# B&R Automation Studio project Palletizer
Automation Studio 4.9

## Logical view

Binary libraries used (declarations not repeated): operator, runtime, astime, AsIecCon, standard, AsArLog, AsBrStr, AsTCP, MTBasics, brsystem, MTTypes, sys_lib, Acp10man, Acp10par, NcGlobal

### Global.var - Global variables
```iecst
(*Feeder*)
(*Inputs*)
VAR
	ResetButton : BOOL;
	laser_sensor_IR : BOOL;
	laser_sensor_2_IR : BOOL;
	carriage_2_AXIS : REAL;
	carriage_2_RCHD : BOOL;
	turnpusher_LBK : BOOL;
	turnpusher_LFR : BOOL;
	pusher_LBK : BOOL;
	pusher_LFR : BOOL;
END_VAR
(*Outputs*)
VAR
	pusher_FW : BOOL;
	conveyor_if_FWD : BOOL;
	conveyor_turn1_FWD : BOOL;
	conveyor_end_FWD : BOOL;
	carrige_2_TGT_POS : REAL;
	turnpusher_FWD : BOOL;
	turnpusher_BWD : BOOL;
END_VAR
(*GenericDevice Feeder requests*)
VAR
	conveyor_if_enable_request : BOOL;
	conveyor_if_disable_request : BOOL;
	conveyor_turn1_enable_request : BOOL;
	conveyor_turn1_disable_request : BOOL;
	conveyor_end_enable_request : BOOL;
	conveyor_end_disable_request : BOOL;
	pusher_enable_request : BOOL;
	pusher_disable_request : BOOL;
	turnpusher_enable_request : BOOL;
	turnpusher_disable_request : BOOL;
	OperationType : INT := 0;
END_VAR
(*Feeder-Main communication variable*)
VAR
	StartMachine : BOOL;
	FeederInitDone : BOOL;
	FeederStart : BOOL;
	FeederHomed : BOOL;
	FeederReady : BOOL;
	FeederEnable : BOOL;
	FeederIsReady : BOOL;
	CraneEnable : BOOL;
	CraneIsReady : BOOL;
	CraneStart : BOOL;
	FeederStop : BOOL;
	vacuum_box_crane_VACUUM : BOOL;
	box_crane_AXIS : REAL;
	gantry_crane_AXIS : REAL;
	gantry_crane_TGT_POS : REAL;
	box_crane_TGT_POS : REAL;
	cardboard_TRIG : BOOL;
	vaccum_box_crane_GRIP : BOOL;
	slide_rail_right_EN : BOOL;
	pusher_z_EN : BOOL;
	pusher_x_EN : BOOL;
END_VAR
(*Crane-Main communication variable*)
VAR
	CraneStop : BOOL;
	CraneHomed : BOOL;
	FeederHoming : BOOL;
	Trigger : BOOL;
	autoreset : BOOL;
	EmergencyStop : BOOL;
	vacuum_box_crane_GRIP : BOOL;
	MainEnable : BOOL;
	MainStart : BOOL;
	PalletHandlerEnable : BOOL;
	pallet_conveyor_2_ACT_VEL : REAL;
	PalletHandlerStart : BOOL;
	pallet_light_barrier_2_IR : BOOL;
	pallet_light_barrier_1_IR : BOOL;
	pallet_conveyor_1_FWD : BOOL;
	pallet_fork_left_EN : BOOL;
	pallet_fork_left_FB : BOOL;
	pallet_lifter_AXIS : REAL;
	pallet_lifter_TGT_POS : REAL;
	PalletHandlerIsReady : BOOL;
	cartboard_TRIG : BOOL;
	PusherXActuatorFaultE : BOOL;
	PusherXDisableSensorFaultE : BOOL;
	PusherXEnableSensorFaultE : BOOL;
	PusherZActuatorFaultE : BOOL;
	PusherZDisableSensorFaultE : BOOL;
	PusherZEnableSensorFaultE : BOOL;
	SlideRailRightActuatorFaultE : BOOL;
	SlideRailRightDisableFaultE : BOOL;
	SlideRailRightEnableFaultE : BOOL;
	VacuumBoxCraneActuatorFaultE : BOOL;
	VacuumBoxCraneDisableFaultE : BOOL;
	VacuumBoxCraneEnableFaultE : BOOL;
	CardboardActuatorFaultE : BOOL;
	CardboardDisableFaultE : BOOL;
	BoxCraneFaultSignalE : BOOL;
	GantryCraneFaultSignalE : BOOL;
	CardboardEnableFaultE : BOOL;
	TurnpusherActuatorFaultE : BOOL;
	TurnpusherDisableSensorFaultE : BOOL;
	TurnpusherEnableSensorFaultE : BOOL;
	PusherActuatorFaultE : BOOL;
	PusherDisableSensorFaultE : BOOL;
	PusherEnableSensorFaultE : BOOL;
	ConveyorIfActuatorFaultE : BOOL;
	ConveyorIfDisableSensorFaultE : BOOL;
	ConveyorIfEnableSensorFaultE : BOOL;
	ConveyorTurn1ActuatorFaultE : BOOL;
	ConveyorTurn1DisableSensorFaultE : BOOL;
	ConveyorTurn1EnableSensorFaultE : BOOL;
	ConveyorEndActuatorFaultE : BOOL;
	ConveyorEndDisableSensorFaultE : BOOL;
	ConveyorEndEnableSensorFaultE : BOOL;
	CarriagePositionFaultSignalE : BOOL;
	PalletForkActuatorFaultE : BOOL;
	PalletForkDisableSensorFaultE : BOOL;
	PalletForkEnableSensorFaultE : BOOL;
	PalletLifterFaultSignalE : BOOL;
	PalletConv1ActuatorFaultE : BOOL;
	PalletConv1DisableSensorFaultE : BOOL;
	PalletConv1SensorFaultE : BOOL;
	PalletConv2FaultSignalE : BOOL;
	LaserSensor2IRFault : BOOL;
	Var2 : BOOL;
	Var1 : BOOL;
	LogFile : STRING[3000];
	MainMessage : STRING[30];
	OnPhaseStop : BOOL;
	ImmediateStop : BOOL;
	ImmediateStopButton : BOOL;
	EmergencyStopButton : BOOL;
	OnPhaseStopPerforming : BOOL;
	OnPhaseStopButton : BOOL;
	laser_sensor_IR_enabled : BOOL;
	pallet_light_barrier_enabled : BOOL;
	laser_sensor_2_IR_enabled : BOOL;
	pallet_light_barrier2_enabled : BOOL;
	InfoCarousel : STRING[20];
	HomeButton : BOOL;
	ErrorButton : BOOL;
	OrangeLight : BOOL;
	YellowLight : BOOL;
	ResetEnable : BOOL;
	WhiteLight : BOOL;
	BlueLight : BOOL;
	GreenLight : BOOL;
	RedLight : BOOL;
	SimPusherActuatorFaultE : BOOL;
	SimPusherDisableSensorFaultE : BOOL;
	SimBoxCraneFaultSignalE : BOOL;
	SimVacuumBoxCraneActuatorFaultE : BOOL;
	SimPalletForkActuatorFaultE : BOOL;
	SimPalletForkEnableSensorFaultE : BOOL;
	OperationTypeString : STRING[20];
	CounterPallet : INT;
END_VAR
```

### Package Logical/Libraries - Global libraries

### Library Logical/Libraries/GenericDev (IEC)

#### Types.typ - Exported data types
```iecst
TYPE
	GenericDeviceStateType :
		(
		DeviceDisabledState,
		DeviceEnablePhaseState,
		DeviceEnabledState,
		DeviceDisablePhaseState
		);
END_TYPE
```

#### Constants.var - Exported constants
```iecst
VAR CONSTANT
	INIT : INT := 0;
	RUN : INT := 1;
	ENABLED : INT := 2;
	STOP : INT := 3;
	DEVICE_WITHOUT_FEEDBACK : INT := 2#01000000;
	DEVICE_WITH_ENABLE_FEEDBACK : INT := 2#00010000;
	DEVICE_WITH_DISABLE_FEEDBACK : INT := 2#00100000;
	DEVICE_WITH_DOUBLE_FEEDBACK : INT := 2#00110000;
	DEVICE_WITH_SINGLE_ACTUATION : INT := 2#00000001;
	DEVICE_WITH_DOUBLE_ACTUATION : INT := 2#00000011;
	DEVICE_IMMEDIATE_STOP_AUTOMATIC : INT := 2#10000000;
	DEVICE_WITH_DA_NO_RETAIN : INT := 2#00000010;
	DEVICE_FEEDBACK_MASK : INT := 2#01110000;
	DEVICE_STOP_MASK : INT := 2#10000000;
	DEVICE_ACTUATION_MASK : INT := 2#00001111;
END_VAR
```

#### GenericDev.fun - Exported functions and function blocks
```iecst
FUNCTION_BLOCK GenericDevice_FB
	VAR_INPUT
		DeviceOperation : INT;
		DeviceType : INT;
		DeviceEnabledSensor : BOOL;
		DeviceDisabledSensor : BOOL;
		DeviceClock : BOOL;
		DeviceEnableTime : INT;
		DeviceDisableTime : INT;
		DeviceDiagnosticsEnabled : BOOL;
		DeviceEnablePreset : BOOL;
		ImmediateStop : BOOL;
	END_VAR
	VAR_OUTPUT
		EnableDevice : BOOL;
		DisableDevice : BOOL;
		DeviceEnabledSensorFault : BOOL;
		DeviceDisabledSensorFault : BOOL;
		DeviceActuatorFault : BOOL;
		DeviceFault : BOOL;
		DeviceNotInitialized : BOOL;
	END_VAR
	VAR_IN_OUT
		DeviceEnableRequest : BOOL;
		DeviceDisableRequest : BOOL;
	END_VAR
	VAR
		DeviceState : GenericDeviceStateType;
		DeviceTimer : INT;
		DeviceTimeout : BOOL;
		DeviceEnabled : BOOL;
		DeviceDisabled : BOOL;
		OldEnableDevice : BOOL;
		Condition : BOOL;
	END_VAR
END_FUNCTION_BLOCK
```

#### GenericDevice_FB.st
```iecst
(*Generic Device function block implementation (See Slide Generic Device)*)
FUNCTION_BLOCK GenericDevice_FB

    // Device clock handler
	IF (DeviceClock AND (DeviceTimer > 0)) THEN
		DeviceTimer := DeviceTimer - 1;
	END_IF;

	// Device sensors handler
	CASE (DeviceType AND DEVICE_FEEDBACK_MASK) OF
		DEVICE_WITH_DISABLE_FEEDBACK:

			DeviceDisabled := DeviceDisabledSensor;

			DeviceEnabled := NOT DeviceDisabled AND
				((DeviceState = DeviceEnabledState) OR
				((DeviceState = DeviceEnablePhaseState) AND DeviceTimeout));

		DEVICE_WITH_ENABLE_FEEDBACK:

			DeviceEnabled := DeviceEnabledSensor;

			DeviceDisabled := NOT DeviceEnabled AND
				((DeviceState = DeviceDisabledState) OR
				((DeviceState = DeviceDisablePhaseState) AND DeviceTimeout));

		DEVICE_WITH_DOUBLE_FEEDBACK:

			DeviceEnabled := DeviceEnabledSensor;

			DeviceDisabled := DeviceDisabledSensor;

		DEVICE_WITHOUT_FEEDBACK:

			DeviceEnabled := (DeviceState = DeviceEnabledState) OR ((DeviceState = DeviceEnablePhaseState) AND DeviceTimeout);

			DeviceDisabled := (DeviceState = DeviceDisabledState) OR ((DeviceState = DeviceDisablePhaseState) AND DeviceTimeout);

	END_CASE;

	// Initialization handler
	IF DeviceOperation = INIT THEN
		CASE (DeviceType AND DEVICE_FEEDBACK_MASK) OF
			DEVICE_WITH_ENABLE_FEEDBACK:
				DeviceDisabled := NOT DeviceEnabled;

			DEVICE_WITH_DISABLE_FEEDBACK:
				DeviceEnabled := NOT DeviceDisabled;

			DEVICE_WITHOUT_FEEDBACK:
				DeviceEnabled := DeviceEnablePreset;
				DeviceDisabled := NOT DeviceEnabled;
		END_CASE;

		DeviceEnableRequest := FALSE;
		DeviceDisableRequest := FALSE;

		IF DeviceEnablePreset THEN
			EnableDevice := TRUE;
			DeviceTimer := DeviceEnableTime;
			IF NOT (DeviceDisabled AND DeviceEnabled) THEN
				DeviceState := DeviceEnablePhaseState;
			ELSE
				DeviceState := DeviceEnabledState;
			END_IF;
			DeviceNotInitialized := NOT DeviceEnabled OR DeviceDisabled;
		ELSE
			EnableDevice := FALSE;
			DeviceTimer := DeviceDisableTime;
			IF NOT (DeviceDisabled AND DeviceEnabled) THEN
				DeviceState := DeviceDisablePhaseState;
			ELSE
				DeviceState := DeviceDisabledState;
			END_IF;
			DeviceNotInitialized := DeviceEnabled OR NOT DeviceDisabled;
		END_IF;
	END_IF;

	// Device control handler (slide 8-9)
	CASE DeviceState OF
		DeviceDisabledState:
			DeviceDisableRequest := FALSE;
			IF (DeviceEnableRequest) THEN
				EnableDevice := TRUE;
				DeviceTimer := DeviceEnableTime;
				DeviceState := DeviceEnablePhaseState;
			END_IF;

		DeviceEnablePhaseState:
			IF (DeviceDisableRequest) THEN
				DeviceEnableRequest := FALSE;
				EnableDevice := FALSE;
				DeviceTimer := DeviceDisableTime;
				DeviceState := DeviceDisablePhaseState;
			END_IF;
			IF (DeviceEnabled) THEN
				DeviceEnableRequest := FALSE;
				//DeviceTimer := 0;
				DeviceState := DeviceEnabledState;
			END_IF;

		DeviceEnabledState:
			DeviceEnableRequest := FALSE;
			IF (DeviceDisableRequest) THEN
				EnableDevice := FALSE;
				DeviceTimer := DeviceDisableTime;
				DeviceState := DeviceDisablePhaseState;
			END_IF;

		DeviceDisablePhaseState:
			IF (DeviceEnableRequest) THEN
				DeviceDisableRequest := FALSE;
				EnableDevice := TRUE;
				DeviceTimer := DeviceEnableTime;
				DeviceState := DeviceEnablePhaseState;
			END_IF;
			IF (DeviceDisabled) THEN
				DeviceDisableRequest := FALSE;
				//DeviceTimer := 0;
				DeviceState := DeviceDisabledState;
			END_IF;
	END_CASE;

	// Device diagnostics handler (slide 26)
	DeviceTimeout := (DeviceTimer = 0);
	IF DeviceDiagnosticsEnabled AND NOT ImmediateStop AND (DeviceType AND DEVICE_FEEDBACK_MASK) <> DEVICE_WITHOUT_FEEDBACK THEN
		CASE (DeviceType AND DEVICE_FEEDBACK_MASK) OF
			DEVICE_WITH_DISABLE_FEEDBACK:

				DeviceDisabledSensorFault :=
				(NOT EnableDevice AND NOT DeviceDisabled AND NOT DeviceEnabled) AND DeviceTimeout;

				DeviceActuatorFault :=
				(EnableDevice AND DeviceDisabled AND NOT DeviceEnabled) AND DeviceTimeout;

			DEVICE_WITH_ENABLE_FEEDBACK:

				DeviceEnabledSensorFault :=
				(EnableDevice AND NOT DeviceDisabled AND NOT DeviceEnabled) AND DeviceTimeout;

				DeviceActuatorFault :=
				(NOT EnableDevice AND NOT DeviceDisabled AND DeviceEnabled) AND DeviceTimeout;

			DEVICE_WITH_DOUBLE_FEEDBACK:

				DeviceDisabledSensorFault :=
				((NOT EnableDevice AND NOT DeviceDisabled AND NOT DeviceEnabled) OR
				(EnableDevice AND DeviceDisabled AND DeviceEnabled)) AND DeviceTimeout;

				DeviceEnabledSensorFault :=
				((NOT EnableDevice AND DeviceDisabled AND DeviceEnabled) OR
				(EnableDevice AND NOT DeviceDisabled AND NOT DeviceEnabled)) AND DeviceTimeout;

				DeviceActuatorFault :=
				((NOT EnableDevice AND NOT DeviceDisabled AND DeviceEnabled) OR
				(EnableDevice AND DeviceDisabled AND NOT DeviceEnabled)) AND DeviceTimeout;

		END_CASE;

		DeviceFault := DeviceDisabledSensorFault OR DeviceEnabledSensorFault OR DeviceActuatorFault;
	END_IF

	IF (DeviceType AND DEVICE_STOP_MASK) = DEVICE_IMMEDIATE_STOP_AUTOMATIC AND ImmediateStop AND NOT Condition THEN
		OldEnableDevice := EnableDevice;
		EnableDevice := FALSE;
		Condition := TRUE;
	ELSIF Condition AND NOT ImmediateStop THEN
		EnableDevice := OldEnableDevice;
		Condition := FALSE;
	END_IF

	// Device actuators handler (correct from slides)
	CASE (DeviceType AND DEVICE_ACTUATION_MASK) OF
		DEVICE_WITH_DOUBLE_ACTUATION:
			DisableDevice := NOT EnableDevice;

		DEVICE_WITH_DA_NO_RETAIN:
			EnableDevice := EnableDevice AND (DeviceState = DeviceEnablePhaseState);
			DisableDevice := NOT EnableDevice AND(DeviceState = DeviceDisablePhaseState);
	END_CASE;

END_FUNCTION_BLOCK
```

### Library Logical/Libraries/GenericAx (IEC)

#### Types.typ - Exported data types
```iecst
TYPE
	GenericAxisStateType :
		(
		CheckCommand,
		WaitTargetPosition,
		WaitTargetVelocity,
		FaultState,
		StopEmergencyState,
		WaitForStop
		);
END_TYPE
```

#### Constants.var - Exported constants
```iecst
VAR CONSTANT
	IDLE : WORD := 0;
	CHANGE_VELOCITY : WORD := 1;
	CHANGE_POSITION : WORD := 2;
	EMERGENCY_STOP_REQUEST : WORD := 3;
	IMMEDIATE_STOP_REQUEST : WORD := 4;
END_VAR
```

#### GenericAx.fun - Exported functions and function blocks
```iecst
{REDUND_ERROR} FUNCTION_BLOCK GenericAxis (*TODO: Add your comment here*) (*$GROUP=User,$CAT=User,$GROUPICON=User.png,$CATICON=User.png*)
	VAR_INPUT
		Command : {REDUND_UNREPLICABLE} WORD := 6;
		ActualPosition : REAL;
		ActualVelocity : REAL;
		NewSetPoint : REAL;
		DeviceTimer : UDINT;
		TGT_SENSOR : BOOL;
		Reset : BOOL;
	END_VAR
	VAR_OUTPUT
		TargetVelocity : REAL;
		TargetPosition : REAL;
		InPosition : BOOL;
		InVelocity : BOOL;
		DeviceFault : BOOL;
	END_VAR
	VAR
		AxisState : GenericAxisStateType;
		Timer : UDINT;
	END_VAR
END_FUNCTION_BLOCK
```

#### GenericAxis.st
```iecst
(* GenericAxis function block *)
FUNCTION_BLOCK GenericAxis

	CASE AxisState OF

		CheckCommand:
			IF Command = CHANGE_POSITION THEN
				IF TargetPosition <> NewSetPoint THEN
					TargetPosition := NewSetPoint;
					InPosition := FALSE;
					Timer := DeviceTimer;
					AxisState := WaitTargetPosition;
				END_IF

			ELSIF Command = CHANGE_VELOCITY THEN
				IF TargetVelocity <> NewSetPoint THEN
					TargetVelocity := NewSetPoint;
					InVelocity := FALSE;
					Timer := DeviceTimer;
					AxisState := WaitTargetVelocity;
				END_IF

			ELSIF Command = IMMEDIATE_STOP_REQUEST OR Command = EMERGENCY_STOP_REQUEST THEN
				TargetPosition := ActualPosition;
				TargetVelocity := 0;
				AxisState := StopEmergencyState;

			ELSIF Command = IDLE THEN
				IF (ActualPosition = TargetPosition AND TGT_SENSOR) THEN
					InPosition := TRUE;
				ELSE
					InPosition := FALSE;
				END_IF
				IF (ActualVelocity = TargetVelocity) THEN
					InVelocity := TRUE;
				ELSE
					InVelocity := FALSE;
				END_IF
				Timer := DeviceTimer;
				DeviceFault := FALSE;
			END_IF

		WaitTargetPosition:
			IF  Command = IMMEDIATE_STOP_REQUEST OR Command = EMERGENCY_STOP_REQUEST THEN
				TargetPosition := ActualPosition;
				TargetVelocity := 0;
				AxisState := StopEmergencyState;
			ELSIF (ActualPosition = TargetPosition AND TGT_SENSOR) THEN
				InPosition := TRUE;
				AxisState := CheckCommand;
			END_IF

			Timer := Timer - 1;
			IF Timer = 0 THEN
				DeviceFault := TRUE;
				AxisState := FaultState;
			END_IF

		WaitTargetVelocity:
			IF  Command = IMMEDIATE_STOP_REQUEST OR Command = EMERGENCY_STOP_REQUEST THEN
				TargetVelocity := 0;
				AxisState := StopEmergencyState;

			ELSIF ActualVelocity = TargetVelocity THEN
				InVelocity := TRUE;
				AxisState := CheckCommand;
			END_IF

			Timer := Timer - 1;
			IF Timer = 0 THEN
				DeviceFault := TRUE;
				AxisState := FaultState;
			END_IF

		StopEmergencyState:
			IF Command <> IMMEDIATE_STOP_REQUEST AND Command <> EMERGENCY_STOP_REQUEST THEN
				InPosition := FALSE;
				InVelocity := FALSE;
				AxisState := CheckCommand;
			END_IF

		FaultState:
			IF Reset THEN
				DeviceFault := FALSE;
				AxisState := CheckCommand;
			END_IF

	END_CASE;

END_FUNCTION_BLOCK
```

### Library Logical/Libraries/Signal_lib (IEC)

#### Constants.var - Exported constants
```iecst
(*OUTPUTS*)
VAR CONSTANT
	NONE : DWORD := 16#0000;
	EMERGENCY_STOP : DWORD := 16#0001;
	ON_PHASE_STOP : DWORD := 16#0010;
	IMMEDIATE_STOP : DWORD := 16#0100; (*Operation types for the Signal Manager*)
	START_CONFIGURATION : USINT := 1;
	CONFIGURATION : USINT := 2;
	START_GENERATION : USINT := 3;
	MESSAGES_GENERATION : USINT := 5;
	GENERATION : USINT := 4; (*SignalCode bitmap*)
	INFORMATION : USINT := 1;
	ANOMALY : USINT := 2;
	WARNING : USINT := 3;
	ALARM : USINT := 4; (*masks for the SiglaCode*)
	DISPLAY_LOG : USINT := 8;
	SIGNAL_TYPE_MASK : USINT := 7;
	SIGNAL_LOG_MASK : USINT := 8;
END_VAR
```

#### Signal_lib.fun - Exported functions and function blocks
```iecst
{REDUND_ERROR} FUNCTION_BLOCK SignalManagement_FB (*TODO: Add your comment here*) (*$GROUP=User,$CAT=User,$GROUPICON=User.png,$CATICON=User.png*)
	VAR_INPUT
		OperationType : INT;
		SignalType : INT; (* bit configuration for the signal*)
		Reset : BOOL;
		KeyReset : BOOL;
		SignalOutput : DWORD; (* Output of the Signal if active*)
		ActivationSignal : {REDUND_UNREPLICABLE} BOOL;
		SignalCode : INT; (* Is the signal number in the priority list*)
		InputString : STRING[80];
	END_VAR
	VAR_OUTPUT
		MainMessage : STRING[30];
		LogFile : STRING[3000];
		SignalOutputs : DWORD; (*Output Signal codification*)
	END_VAR
	VAR
		LogBuffer : ARRAY[1..100] OF STRING[30];
		NumberOfAlarms : INT; (*Counters*)
		NumberOfAnomalies : INT;
		NumberOfWarnings : INT;
		NumberOfInformation : INT; (*Counters for Active Signals*)
		NumberOfActiveAlarms : INT;
		NumberOfActiveAnomalies : INT;
		NumberOfActiveWarning : INT;
		NumberOfActiveInformation : INT; (*Reset Management*)
	END_VAR
	VAR_OUTPUT
		ResetEnable : BOOL;
	END_VAR
	VAR
		ResetActivation : BOOL;
		AuxResetActivation : BOOL;
		Signals : ARRAY[1..100] OF BOOL; (*Signals management*)
		ActiveSignalCodes : ARRAY[1..100] OF INT;
		ResetOld : BOOL; (*Auxiliary variable*)
		KeyResetOld : BOOL;
		Index : INT;
		BaseIndex : INT;
		Condition : BOOL;
		i : INT;
	END_VAR
END_FUNCTION_BLOCK
```

#### SignalManagement_FB.st
```iecst
(* TODO: Add your comment here *)
FUNCTION_BLOCK SignalManagement_FB

	CASE OperationType OF
		START_CONFIGURATION:  (* Reset signals counts *)
			NumberOfAlarms := 0;
			NumberOfAnomalies := 0;
			NumberOfWarnings := 0;
			NumberOfInformation := 0;
			ResetEnable := FALSE;
		CONFIGURATION:
			(* counting signals *)
			CASE SignalType AND SIGNAL_TYPE_MASK OF
				ALARM:
					NumberOfAlarms := NumberOfAlarms + 1;
				ANOMALY:
					NumberOfAnomalies := NumberOfAnomalies + 1;
				WARNING:
					NumberOfWarnings := NumberOfWarnings + 1;
				INFORMATION:
					NumberOfInformation := NumberOfInformation + 1;
			END_CASE
		START_GENERATION:
			(* Prepare for generation *)
			ResetEnable := FALSE;
			SignalOutputs := NONE;
			ResetActivation := Reset AND NOT ResetOld;
			ResetOld := Reset;
			AuxResetActivation := KeyReset AND NOT KeyResetOld;
			KeyResetOld:= KeyReset;
			LogFile := '';
			MainMessage := '';

		GENERATION:
			CASE SignalType AND SIGNAL_TYPE_MASK OF
				ALARM:
					Index := NumberOfActiveAlarms;
					BaseIndex := 0;
					Condition := TRUE;
				ANOMALY:
					Index := NumberOfActiveAnomalies;
					BaseIndex := NumberOfAlarms;
					Condition := TRUE;
				WARNING:
					Index := NumberOfActiveWarning;
					BaseIndex := NumberOfAlarms + NumberOfAnomalies;
					Condition := FALSE;
				INFORMATION:
					Index := NumberOfActiveInformation;
					BaseIndex := NumberOfAlarms + NumberOfAnomalies + NumberOfWarnings;
					Condition := FALSE;
			END_CASE
			IF ActivationSignal AND NOT Signals[SignalCode] THEN
				Signals[SignalCode] := TRUE;
				Index := Index + 1;
				ActiveSignalCodes[BaseIndex + Index] := SignalCode;

				IF (SignalType AND SIGNAL_LOG_MASK) = DISPLAY_LOG THEN
					LogBuffer[SignalCode] := InputString;
				END_IF

			END_IF
			IF Condition AND Signals[SignalCode] AND NOT ActivationSignal AND (ActiveSignalCodes[BaseIndex + 1] = SignalCode) THEN
				ResetEnable := TRUE;
			END_IF

			IF (ResetActivation OR NOT Condition) AND Signals[SignalCode] AND NOT ActivationSignal AND (ActiveSignalCodes[BaseIndex + 1] = SignalCode) THEN
				Signals[SignalCode] := FALSE;
				FOR i := 2 TO Index DO
					ActiveSignalCodes[BaseIndex + i-1] := ActiveSignalCodes[BaseIndex + i];
				END_FOR;
				ActiveSignalCodes[BaseIndex + Index] := 0;
				Index :=  Index - 1;
				ResetActivation := FALSE; (* COMMENT THIS LINE TO GO BACK TO CUMULATIVE RESET *)

				IF (SignalType AND SIGNAL_LOG_MASK) = DISPLAY_LOG THEN
					LogBuffer[SignalCode] := ' ';
				END_IF

			END_IF
			CASE SignalType AND SIGNAL_TYPE_MASK OF
				ALARM:
					NumberOfActiveAlarms := Index;
				ANOMALY:
					NumberOfActiveAnomalies := Index;
				WARNING:
					NumberOfActiveWarning := Index;
				INFORMATION:
					NumberOfActiveInformation := Index;
			END_CASE
			IF Signals[SignalCode] THEN
				SignalOutputs := SignalOutputs OR SignalOutput;
			END_IF

		MESSAGES_GENERATION:

			LogFile := ' ';
			// ALARMS messages creation
			BaseIndex := 0;
			FOR i := 1 TO NumberOfActiveAlarms DO
				IF LogBuffer[ActiveSignalCodes[BaseIndex + i]] <> '' THEN
					LogFile := CONCAT(CONCAT(LogFile, CONCAT('ALARM : ',LogBuffer[ActiveSignalCodes[BaseIndex + i]])), ' \n ');
				END_IF
			END_FOR;

			// ANOMALIES messages creation
			BaseIndex := NumberOfAlarms;
			FOR i := 1 TO NumberOfActiveAnomalies DO
				IF LogBuffer[ActiveSignalCodes[BaseIndex + i]] <> '' THEN
					LogFile := CONCAT(CONCAT(LogFile,CONCAT('ANOMALY : ',LogBuffer[ActiveSignalCodes[BaseIndex + i]])), ' \n ');
				END_IF

			END_FOR;

			// WARNING messages creation
			BaseIndex := NumberOfAlarms + NumberOfAnomalies;
			FOR i := 1 TO NumberOfActiveWarning DO
				IF LogBuffer[ActiveSignalCodes[BaseIndex + i]] <> '' THEN
					LogFile := CONCAT(CONCAT(LogFile , CONCAT('WARNING : ',LogBuffer[ActiveSignalCodes[BaseIndex + i]])), ' \n ');
				END_IF
			END_FOR;

			// WARNING messages creation
			BaseIndex := NumberOfAlarms + NumberOfAnomalies + NumberOfWarnings;
			FOR i := 1 TO NumberOfActiveInformation DO
				IF LogBuffer[ActiveSignalCodes[BaseIndex + i]] <> '' THEN
					LogFile := CONCAT(CONCAT(LogFile , CONCAT('INFORMATION : ',LogBuffer[ActiveSignalCodes[BaseIndex + i]])), ' \n ');
				END_IF
			END_FOR;

			MainMessage := '';
			IF NumberOfActiveAlarms <> 0 THEN
				MainMessage := LogBuffer[ActiveSignalCodes[1]];
			ELSIF NumberOfActiveAnomalies <> 0 THEN
				MainMessage := LogBuffer[ActiveSignalCodes[NumberOfAlarms + 1]];
			ELSIF NumberOfActiveWarning <> 0 THEN
				MainMessage := LogBuffer[ActiveSignalCodes[NumberOfAlarms + NumberOfAnomalies + 1]];
			ELSIF NumberOfActiveInformation <> 0 THEN
				MainMessage := LogBuffer[ActiveSignalCodes[NumberOfAlarms + NumberOfAnomalies + NumberOfWarnings + 1]];
			END_IF

	END_CASE

END_FUNCTION_BLOCK
```

### Library Logical/Libraries/Filter (IEC)

#### Filter.fun - Exported functions and function blocks
```iecst
{REDUND_ERROR} {REDUND_UNREPLICABLE} FUNCTION_BLOCK filter_FB (*TODO: Add your comment here*) (*$GROUP=User,$CAT=User,$GROUPICON=User.png,$CATICON=User.png*)
	VAR_INPUT
		OperationType : {REDUND_UNREPLICABLE} INT;
		Clock : {REDUND_UNREPLICABLE} BOOL;
		Signal : {REDUND_UNREPLICABLE} BOOL;
		DeactivationDelay : {REDUND_UNREPLICABLE} INT;
		ActivationDelay : {REDUND_UNREPLICABLE} INT;
	END_VAR
	VAR_OUTPUT
		DelayedSignal : {REDUND_UNREPLICABLE} BOOL;
	END_VAR
	VAR
		Delay : {REDUND_UNREPLICABLE} INT;
	END_VAR
END_FUNCTION_BLOCK
```

#### filter_FB.st
```iecst
(* TODO: Add your comment here *)
FUNCTION_BLOCK filter_FB

	IF (OperationType = INIT) THEN
		Delay := 0;
	END_IF;

	IF (Clock AND (Delay > 0)) THEN
		Delay := Delay - 1;
	END_IF;

	IF  (Delay = 0) THEN
		DelayedSignal := Signal;
	END_IF;

	IF  (Signal = DelayedSignal) THEN
		IF  (Signal) THEN
			Delay := DeactivationDelay;
		ELSE
			Delay := ActivationDelay;
		END_IF;
	END_IF

END_FUNCTION_BLOCK
```

### Program Logical/MainCtrl (IEC)

#### Types.typ
```iecst
TYPE
	MainStateType :
		(
		Idle,
		Ready,
		Run,
		Init
		);
END_TYPE
```

#### Variables.var
```iecst
VAR
	MachineState : MainStateType;
END_VAR
```

#### Main.st
```iecst
PROGRAM _INIT

		MachineState := Idle;
END_PROGRAM

PROGRAM _CYCLIC

	CASE MachineState OF

		Idle:
			FeederEnable := FALSE;
			FeederHomed := FALSE;
			FeederStart := FALSE;

			IF StartMachine THEN
				FeederEnable := TRUE; (* sblocca alimentazione feeder *)
				MachineState := Init;
			END_IF

		Init:
			OperationType := INIT;
			StartMachine := FALSE;
			//FeederHomed := TRUE; (* manda homing feeder *)
			IF FeederHomed THEN // Need to add also the carriage
				FeederInitDone := TRUE;
			END_IF

			// Perform the same procedure for all the other 3 machines
			IF FeederInitDone THEN
				FeederReady := TRUE;  // States that all 3 machines are ready (now we consider only the feeder)
			END_IF

			IF FeederReady THEN
				MachineState := Ready;
			END_IF
		Ready:
			(* Attesa che anche crane e pallet handler siano ready, ora non li abbiamo *)
			OperationType := READY;
			IF StartMachine THEN
				FeederStart := TRUE;
				MachineState := Run;
			END_IF
		Run:
			OperationType := RUN;
			FeederHomed := FALSE;
			FeederEnable := TRUE;
			FeederStart := TRUE;

	END_CASE

END_PROGRAM

PROGRAM _EXIT
	(* Insert code here *)

END_PROGRAM
```

### MNG_Global.typ - Global data types
```iecst
(* 3d position *)

TYPE
	VEC3 : 	STRUCT
		x : REAL;
		y : REAL;
		z : REAL;
	END_STRUCT;
END_TYPE

(* position and orientation as an euler based pose *)

TYPE
	POSE6 : 	STRUCT
		x : REAL;
		y : REAL;
		z : REAL;
		a : REAL;
		b : REAL;
		c : REAL;
	END_STRUCT;
END_TYPE

(* position and orientation as a 4x4 matrix *)

TYPE
	TRAFO : 	STRUCT
		baseX : VEC3;
		fill0 : REAL;
		baseY : VEC3;
		fill1 : REAL;
		baseZ : VEC3;
		fill2 : REAL;
		origin : VEC3;
		fill3 : REAL;
	END_STRUCT;
END_TYPE
```

### Program Logical/FeederMachine (IEC)

#### Types.typ
```iecst
TYPE
	StateType :
		(
		Idle,
		EnableDone,
		Homing,
		HomingDone,
		WaitForStart,
		WaitForBoxes,
		PushBox,
		CheckSecondLaser,
		CheckPusherBackwardPosition,
		WaitBeforeCarriage,
		CarriageMidPush,
		CarriageTotalPush,
		CarriagePushBack,
		CarriageWaitForStart,
		EmergencyState,
		StopState,
		ImmediateStopState,
		CarriageMidPushDone,
		CarriageTotalPushDone
		);
END_TYPE
```

#### Variables.var
```iecst
VAR
	State : StateType;
END_VAR
(*Generic device variable interface for on/off actuations*)
(*conveyor_if*)
VAR
	conveyor_if : GenericDevice_FB;
END_VAR
VAR CONSTANT
	conveyor_if_enable_time : INT := 5;
	conveyor_if_disable_time : INT := 5;
END_VAR
VAR
	conveyor_if_enable_request : BOOL;
	conveyor_if_disable_request : BOOL;
END_VAR
(*conveyot_turn1*)
VAR
	conveyor_turn1 : GenericDevice_FB;
END_VAR
VAR CONSTANT
	conveyor_turn1_enable_time : INT := 5;
	conveyor_turn1_disable_time : INT := 5;
END_VAR
VAR
	conveyor_turn1_enable_request : BOOL;
	conveyor_turn1_disable_request : BOOL;
END_VAR
(*conveyor_end*)
VAR
	conveyor_end : GenericDevice_FB;
END_VAR
VAR CONSTANT
	conveyor_end_enable_time : INT := 5;
	conveyor_end_disable_time : INT := 5;
END_VAR
VAR
	conveyor_end_enable_request : BOOL;
	conveyor_end_disable_request : BOOL;
END_VAR
(*pusher*)
VAR
	pusher : GenericDevice_FB;
END_VAR
VAR CONSTANT
	pusher_enable_time : INT := 200;
	pusher_disable_time : INT := 200;
END_VAR
VAR
	pusher_enable_request : BOOL;
	pusher_disable_request : BOOL;
END_VAR
(*turnpusher*)
VAR
	turnpusher : GenericDevice_FB;
END_VAR
VAR CONSTANT
	turnpusher_enable_time : INT := 200;
	turnpusher_disable_time : INT := 200;
END_VAR
VAR
	turnpusher_enable_request : BOOL;
	turnpusher_disable_request : BOOL;
END_VAR
(*carriage*)
VAR
	carriage : GenericAxis;
	carriage_goal : REAL;
END_VAR
VAR CONSTANT
	carriage_timer : INT := 100;
END_VAR
VAR
	carriagePositionReached : BOOL;
	carriageSetPoint : USINT;
	carriage_homed : BOOL;
END_VAR
VAR CONSTANT
	HOME_POSITION : REAL := 0.0;
	CARRIAGE_MID_PUSH : REAL := 0.44;
	CARRIAGE_TOTAL_PUSH : REAL := 1.11;
END_VAR
(*Insert your comment here.*)
VAR
	CounterBox : {REDUND_UNREPLICABLE} INT := 0;
	CounterLayer : INT;
	CounterFloor : INT;
	BoxNumber : INT;
	LayerNumber : INT;
END_VAR
(*Fault Laser sensors management*)
VAR CONSTANT
	LaserSensorIRTimer : INT := 10;
END_VAR
VAR
	LaserSensorIRFault : BOOL;
END_VAR
VAR CONSTANT
	LaserSensor2IRTimer : INT := 10;
END_VAR
VAR
	OldState : StateType;
	EmergencyStopMachine : INT;
	ImmediateStopMachine : INT;
	SuspendDevices : BOOL;
	OldPositionCarriageGoal : REAL;
	OldCarriageCommand : WORD;
END_VAR
```

#### Main.st
```iecst
// FEEDER MACHINE
// INTERFACE
// 	INPUT:
// 		FeederEnable : BOOL : It enables the machine and executes the Homing if it is not already done.
//		FeederStart : BOOL : It starts a machine cycle if The machine is Ready
//		FeederStop : BOOL
//		FeederEmergencyStop : BOOL
//
//	OUTPUT:
//		FeederIsEnable : BOOL : True if the machine is ready to start a new cycle.
//		FeederIsReady : BOOL : True if the machine is ready to start a new cycle.
//		FeederIsStop : BOOL
//		FeederIsStopEmergency : BOOL

PROGRAM _INIT
	(* Insert code here *)
	State := Idle;

	CounterBox := 0;	// Box Counter
	CounterLayer := 0;	// Layer Counter
	CounterFloor := 1;	// Starting the counter from Floor 1 due to the MOD operator
	BoxNumber := 8; 	// Start with 8 boxes (turnpuher disabled)
	LayerNumber := 3; 	// Number of layer in a Floor

	// Output requests initialization
	pusher_enable_request := FALSE;
	pusher_disable_request := FALSE;
	turnpusher_enable_request := FALSE;
	turnpusher_disable_request := FALSE;
	conveyor_if_enable_request := FALSE;
	conveyor_if_disable_request := FALSE;
	conveyor_turn1_enable_request := FALSE;
	conveyor_turn1_disable_request := FALSE;
	conveyor_end_enable_request := FALSE;
	conveyor_end_disable_request := FALSE;
	carriage.Command := IDLE;
	//Fault
	LaserSensorIRFault := FALSE;
	LaserSensor2IRFault := FALSE;

	carriage_homed := FALSE;
END_PROGRAM

PROGRAM _CYCLIC

	CASE EmergencyStopMachine OF
		0:
			IF EmergencyStop AND State <> EmergencyState THEN
				State := EmergencyState;
				conveyor_if_disable_request := TRUE;
				conveyor_turn1_disable_request := TRUE;
				conveyor_end_disable_request := TRUE;
				carriage.Command := EMERGENCY_STOP_REQUEST;
				EmergencyStopMachine := 1;
			END_IF

		1:
			IF NOT EmergencyStop THEN
				EmergencyStopMachine := 0;
			END_IF
	END_CASE

	CASE ImmediateStopMachine OF
		0:
			IF ImmediateStop AND State <> ImmediateStopState THEN
				OldState := State;
				SuspendDevices := TRUE;
				OldCarriageCommand := carriage.Command;
				OldPositionCarriageGoal := carriage_goal;
				carriage.Command := IMMEDIATE_STOP_REQUEST;
				State := ImmediateStopState;
				ImmediateStopMachine := 1;
			END_IF

		1:
			IF NOT ImmediateStop THEN
				ImmediateStopMachine := 0;
			END_IF
	END_CASE

	CASE State OF
		EmergencyState:
			IF NOT EmergencyStop THEN
				FeederIsReady := FALSE;
				FeederEnable := FALSE;
				carriage.Command := IDLE;
				State := Idle;
			END_IF

		ImmediateStopState:
			IF NOT ImmediateStop AND FeederStart THEN
				FeederStart := FALSE;
				SuspendDevices := FALSE;
				State := OldState;
				carriage.Command := OldCarriageCommand;
				carriage_goal := OldPositionCarriageGoal;
			END_IF

		Idle:
			IF FeederEnable THEN
				State := Homing;
				pusher_disable_request := TRUE;
				turnpusher_disable_request := TRUE;
				CounterBox := 0;
				CounterLayer := 0;
				CounterFloor := 1;
				BoxNumber := 8;
				LayerNumber := 3;
				// comando di homing carriage solo se serve --- DA VEDERE
				IF carriage.ActualPosition <> HOME_POSITION THEN
					carriage.Command := CHANGE_POSITION;
					carriage_goal := HOME_POSITION;
				END_IF
			END_IF

		Homing:
			IF pusher_disable_request = FALSE AND turnpusher_disable_request = FALSE AND carriagePositionReached THEN
				OldPositionCarriageGoal := carriage_goal;
				OldCarriageCommand := carriage.Command;
				conveyor_if_enable_request := FALSE;
				conveyor_if_disable_request := FALSE;
				carriage.Command := IDLE;
				FeederIsReady := TRUE;
				FeederEnable := FALSE;
				State := HomingDone;
			END_IF

		HomingDone:
			// feeder ready, ora aspetta start
			IF FeederStart THEN
				FeederStart := FALSE;
				FeederIsReady := FALSE;
				CounterLayer := 0;
				State := WaitForStart;
			END_IF

		WaitForStart:
			// counter reset at each cycle
			IF carriagePositionReached THEN
				CounterBox := 0;
				State := WaitForBoxes;
				conveyor_if_enable_request := TRUE;
				conveyor_turn1_enable_request := TRUE;
				conveyor_end_enable_request := TRUE;
			END_IF

		WaitForBoxes:
			IF conveyor_if_enable_request = FALSE
				AND conveyor_turn1_enable_request = FALSE
				AND conveyor_end_enable_request = FALSE THEN

				IF laser_sensor_IR_enabled THEN
					FeederHomed := FALSE;
					State := PushBox;
					conveyor_if_disable_request := TRUE;
					pusher_enable_request := TRUE;
				END_IF

			END_IF

		PushBox:
			IF pusher_enable_request = FALSE AND conveyor_if_disable_request = FALSE THEN
				State := CheckSecondLaser;
			END_IF

		CheckSecondLaser:
			IF laser_sensor_2_IR_enabled THEN
				CounterBox := CounterBox + 1;
				State := CheckPusherBackwardPosition;
				pusher_disable_request := TRUE;
			END_IF

		CheckPusherBackwardPosition:
			IF pusher_disable_request = FALSE THEN
				IF CounterBox < BoxNumber THEN
					conveyor_if_enable_request := TRUE;
					State := WaitForBoxes;
				ELSE
					CounterLayer := CounterLayer + 1;
					conveyor_turn1_disable_request := TRUE;
					conveyor_end_disable_request := TRUE;
					State := WaitBeforeCarriage;
				END_IF
			END_IF

		WaitBeforeCarriage:
			IF conveyor_turn1_disable_request = FALSE AND conveyor_end_disable_request = FALSE THEN
				IF CounterLayer < LayerNumber THEN
					carriage.Command := CHANGE_POSITION;
					carriage_goal := CARRIAGE_MID_PUSH;
					State := CarriageMidPush;
				ELSE
					FeederIsReady := TRUE;
					State := CarriageWaitForStart;
				END_IF
			END_IF

		CarriageWaitForStart:
			IF FeederStart THEN
				FeederStart := FALSE;
				FeederIsReady := FALSE;
				carriage.Command := CHANGE_POSITION;
				carriage_goal := CARRIAGE_TOTAL_PUSH;
				State := CarriageTotalPush;
			END_IF

		CarriageMidPush:
			IF carriagePositionReached THEN
				IF (CounterFloor MOD 2 = 1) = TRUE THEN
					IF CounterLayer > 0 THEN
						turnpusher_enable_request := TRUE;
						turnpusher_disable_request := FALSE;
						BoxNumber := 3;
					ELSE
						turnpusher_enable_request := FALSE;
						turnpusher_disable_request := TRUE;
						BoxNumber := 8;
					END_IF
				ELSE
					IF CounterLayer > 1 THEN
						turnpusher_enable_request := FALSE;
						turnpusher_disable_request := TRUE;
						BoxNumber := 8;
					ELSE
						turnpusher_enable_request := TRUE;
						turnpusher_disable_request := FALSE;
						BoxNumber := 3;
					END_IF
				END_IF

				State := CarriagePushBack;
			END_IF

		CarriageTotalPush:
			IF carriagePositionReached AND turnpusher_enable_request = FALSE AND turnpusher_disable_request = FALSE THEN
				CounterFloor := CounterFloor + 1;
				State := CarriagePushBack;
			END_IF

		CarriagePushBack:
			IF carriagePositionReached THEN
				carriage.Command := CHANGE_POSITION;
				carriage_goal := HOME_POSITION;
				IF CounterLayer = 3 THEN
					State := HomingDone;
					FeederIsReady := TRUE;
				ELSE
					State := WaitForStart;
				END_IF
			END_IF

	END_CASE;

	// DEVICE CALLS

	// pusher
	pusher.DeviceOperation := OperationType;
	pusher.DeviceClock := TRUE;
	pusher.DeviceDiagnosticsEnabled := TRUE;
	pusher.DeviceEnablePreset := FALSE;
	pusher.DeviceEnableTime := pusher_enable_time;
	pusher.DeviceDisableTime := pusher_disable_time;
	pusher.DeviceType := DEVICE_WITH_DOUBLE_FEEDBACK OR DEVICE_WITH_SINGLE_ACTUATION;
	pusher.DeviceEnabledSensor := pusher_LFR;
	pusher.DeviceDisabledSensor := pusher_LBK;
	pusher(DeviceEnableRequest := pusher_enable_request, DeviceDisableRequest := pusher_disable_request);
	pusher_FW := pusher.EnableDevice;

	// turnpusher
	turnpusher.DeviceOperation := OperationType;
	turnpusher.DeviceClock := TRUE;
	turnpusher.DeviceDiagnosticsEnabled := TRUE;
	turnpusher.DeviceEnablePreset := FALSE;
	turnpusher.DeviceEnableTime := turnpusher_enable_time;
	turnpusher.DeviceDisableTime := turnpusher_disable_time;
	turnpusher.DeviceType := DEVICE_WITH_DOUBLE_FEEDBACK OR DEVICE_WITH_DOUBLE_ACTUATION;
	turnpusher.DeviceEnabledSensor := turnpusher_LFR;
	turnpusher.DeviceDisabledSensor := turnpusher_LBK;
	turnpusher(DeviceEnableRequest := turnpusher_enable_request, DeviceDisableRequest := turnpusher_disable_request);
	turnpusher_FWD := turnpusher.EnableDevice;
	turnpusher_BWD := turnpusher.DisableDevice;

	// conveyor_if
	conveyor_if.DeviceOperation := OperationType;
	conveyor_if.DeviceClock := TRUE;
	conveyor_if.DeviceDiagnosticsEnabled := TRUE;
	conveyor_if.ImmediateStop := SuspendDevices OR EmergencyStop;
	conveyor_if.DeviceEnablePreset := FALSE;
	conveyor_if.DeviceEnableTime := conveyor_if_enable_time;
	conveyor_if.DeviceDisableTime := conveyor_if_disable_time;
	conveyor_if.DeviceType := DEVICE_WITHOUT_FEEDBACK OR DEVICE_WITH_SINGLE_ACTUATION OR DEVICE_IMMEDIATE_STOP_AUTOMATIC;
	conveyor_if(DeviceEnableRequest := conveyor_if_enable_request, DeviceDisableRequest := conveyor_if_disable_request);
	conveyor_if_FWD := conveyor_if.EnableDevice;

	// conveyor_turn1
	conveyor_turn1.DeviceOperation := OperationType;
	conveyor_turn1.DeviceClock := TRUE;
	conveyor_turn1.DeviceDiagnosticsEnabled := TRUE;
	conveyor_turn1.ImmediateStop := SuspendDevices OR EmergencyStop;
	conveyor_turn1.DeviceEnablePreset := FALSE;
	conveyor_turn1.DeviceEnableTime := conveyor_turn1_enable_time;
	conveyor_turn1.DeviceDisableTime := conveyor_turn1_disable_time;
	conveyor_turn1.DeviceType := DEVICE_WITHOUT_FEEDBACK OR DEVICE_WITH_SINGLE_ACTUATION OR DEVICE_IMMEDIATE_STOP_AUTOMATIC;
	conveyor_turn1(DeviceEnableRequest := conveyor_turn1_enable_request, DeviceDisableRequest := conveyor_turn1_disable_request);
	conveyor_turn1_FWD := conveyor_turn1.EnableDevice;

	// conveyor_end
	conveyor_end.DeviceOperation := OperationType;
	conveyor_end.DeviceClock := TRUE;
	conveyor_end.DeviceDiagnosticsEnabled := TRUE;
	conveyor_end.ImmediateStop := SuspendDevices OR EmergencyStop;
	conveyor_end.DeviceEnablePreset := FALSE;
	conveyor_end.DeviceEnableTime := conveyor_end_enable_time;
	conveyor_end.DeviceDisableTime := conveyor_end_disable_time;
	conveyor_end.DeviceType := DEVICE_WITHOUT_FEEDBACK OR DEVICE_WITH_SINGLE_ACTUATION OR DEVICE_IMMEDIATE_STOP_AUTOMATIC;
	conveyor_end(DeviceEnableRequest := conveyor_end_enable_request, DeviceDisableRequest := conveyor_end_disable_request);
	conveyor_end_FWD := conveyor_end.EnableDevice;

	// carriage
	carriage.NewSetPoint := carriage_goal;
	carriage.DeviceTimer := carriage_timer; // if elapsed gives fault (See GenericAxis library)
	carriage.ActualPosition := carriage_2_AXIS;
	carriage.TGT_SENSOR := carriage_2_RCHD;
	carrige_2_TGT_POS := carriage.TargetPosition;
	carriagePositionReached := carriage.InPosition;
	carriage();

	// Signals

	// turnpusher fault signals (TO BE DEFINED AS GLOBAL VARIABLES)
	TurnpusherActuatorFaultE := turnpusher.DeviceActuatorFault;
	TurnpusherDisableSensorFaultE := turnpusher.DeviceDisabledSensorFault;
	TurnpusherEnableSensorFaultE := turnpusher.DeviceEnabledSensorFault;

	// pusher fault signals (TO BE DEFINED AS GLOBAL VARIABLES)
	PusherActuatorFaultE := pusher.DeviceActuatorFault;
	PusherDisableSensorFaultE := pusher.DeviceDisabledSensorFault;
	PusherEnableSensorFaultE := pusher.DeviceEnabledSensorFault;

	// conveyor_if fault signals (TO BE DEFINED AS GLOBAL VARIABLES)
	ConveyorIfActuatorFaultE := conveyor_if.DeviceActuatorFault;
	ConveyorIfDisableSensorFaultE := conveyor_if.DeviceDisabledSensorFault;
	ConveyorIfEnableSensorFaultE := conveyor_if.DeviceEnabledSensorFault;

	// conveyor_turn1 fault signals (TO BE DEFINED AS GLOBAL VARIABLES)
	ConveyorTurn1ActuatorFaultE := conveyor_turn1.DeviceActuatorFault;
	ConveyorTurn1DisableSensorFaultE := conveyor_turn1.DeviceDisabledSensorFault;
	ConveyorTurn1EnableSensorFaultE := conveyor_turn1.DeviceEnabledSensorFault;

	// conveyor_end fault signals (TO BE DEFINED AS GLOBAL VARIABLES)
	ConveyorEndActuatorFaultE := conveyor_end.DeviceActuatorFault;
	ConveyorEndDisableSensorFaultE := conveyor_end.DeviceDisabledSensorFault;
	ConveyorEndEnableSensorFaultE := conveyor_end.DeviceEnabledSensorFault;

	// carriage fault signals (TO BE DEFINED AS GLOBAL VARIABLES)
	CarriagePositionFaultSignalE := carriage.DeviceFault;

END_PROGRAM

PROGRAM _EXIT
	(* Insert code here *)
END_PROGRAM
```

### Program Logical/CraneMachine (IEC)

#### Types.typ
```iecst
TYPE
	StateType :
		(
		Idle,
		CardBoardPickHoming,
		CardBoardVacuumHoming,
		Homing,
		HomingDone,
		MoveToCardBoardPositioning,
		CardBoardPositioning,
		MoveToPallet,
		FreeBoxes,
		MoveToCardBoardBuffer1,
		MoveToCardBoardBuffer2_1,
		MoveToCardBoardBuffer2_2,
		CardBoardPick,
		MoveToHomingPosition,
		CheckForHomingDone,
		SetUp,
		CardBoardVacuum,
		EmergencyState,
		StopState,
		ImmediateStopState
		);
END_TYPE
```

#### Variables.var
```iecst
(*box_crane*)
VAR
	box_crane : GenericAxis;
END_VAR
VAR CONSTANT
	BOX_CRANE_HOMING_POSITION : REAL := 0.0;
	BOX_CRANE_FLOOR1_POSITION : REAL := -0.2;
	BOX_CRANE_FLOOR2_POSITION : REAL := 0.01;
	CARDBOARD_PICK_POSITION : REAL := -0.195;
END_VAR
VAR
	BoxCranePositionReached : BOOL;
	box_crane_goal : REAL;
END_VAR
VAR CONSTANT
	box_crane_timer : INT := 200;
END_VAR
(*gantry_crane*)
VAR
	gantry_crane : GenericAxis;
END_VAR
VAR CONSTANT
	GANTRY_CRANE_HOMING_POSITION : REAL := 0.0;
	GANTRY_CRANE_CARDBOARD_POSITION : REAL := -1.11;
	GANTRY_CRANE_PALLET_POSITION : REAL := -1.3;
END_VAR
VAR
	GantryCranePositionReached : BOOL;
	gantry_crane_goal : REAL;
END_VAR
VAR CONSTANT
	gantry_crane_timer : INT := 200;
END_VAR
(*pusher_x request*)
VAR
	pusher_x : GenericDevice_FB;
	pusher_x_enable_request : BOOL;
	pusher_x_disable_request : BOOL;
END_VAR
VAR CONSTANT
	pusher_x_enable_time : INT := 5;
	pusher_x_disable_time : INT := 5;
END_VAR
(*pusher_z request*)
VAR
	pusher_z : GenericDevice_FB;
	pusher_z_enable_request : BOOL;
	pusher_z_disable_request : BOOL;
END_VAR
VAR CONSTANT
	pusher_z_enable_time : INT := 5;
	pusher_z_disable_time : INT := 5;
END_VAR
(*slide_rail_right request*)
VAR
	slide_rail_right : GenericDevice_FB;
	slide_rail_right_enable_request : BOOL;
	slide_rail_right_disable_request : BOOL;
END_VAR
VAR CONSTANT
	slide_rail_right_enable_time : INT := 10;
	slide_rail_right_disable_time : INT := 10;
END_VAR
(*vacuum_box_crane request*)
VAR
	vacuum_box_crane : GenericDevice_FB;
	vacuum_box_crane_enable_request : BOOL;
	vacuum_box_crane_disable_request : BOOL;
END_VAR
VAR CONSTANT
	vacuum_box_crane_enable_time : INT := 200;
	vacuum_box_crane_disable_time : INT := 5;
END_VAR
(*cardboard*)
VAR
	cardboard : GenericDevice_FB;
	cardboard_enable_request : BOOL;
	cardboard_disable_request : BOOL;
END_VAR
VAR CONSTANT
	cardboard_enable_time : INT := 5;
	cardboard_disable_time : INT := 5;
END_VAR
VAR
	State : StateType;
	CounterFloor : INT;
	EmergencyStopMachine : INT;
	ImmediateStopMachine : INT;
	OldState : StateType;
	OldBoxCraneCommand : WORD;
	OldGantryCraneCommand : WORD;
	OldPositionBoxCraneGoal : REAL;
	OldPositionGantryCraneGoal : REAL;
END_VAR
```

#### Main.st
```iecst
// CRANE MACHINE
// INTERFACE
// 	INPUT:
// 		CraneEnable : BOOL : It enables the machine and executes the Homing if it is not already done.
//		CraneStart : BOOL : It starts a machine cycle if The machine is Ready
//		CraneStop : BOOL
//		CraneEmergencyStop : BOOL
//
//	OUTPUT:
//		CraneIsEnable : BOOL : True if the machine is ready to start a new cycle.
//		CraneIsReady : BOOL : True if the machine is ready to start a new cycle.
//		CraneIsStop : BOOL
//		CraneIsStopEmergency : BOOL

PROGRAM _INIT
	(* Insert code here *)
	State := Idle;

	pusher_x_enable_request := FALSE;
	pusher_x_disable_request := FALSE;
	pusher_z_enable_request := FALSE;
	pusher_z_disable_request := FALSE;
	slide_rail_right_enable_request := FALSE;
	slide_rail_right_disable_request := FALSE;
	vacuum_box_crane_enable_request := FALSE;
	vacuum_box_crane_disable_request := FALSE;
	cardboard_enable_request := FALSE;
	cardboard_disable_request := FALSE;

	CounterFloor := 0;
	box_crane.Command := IDLE;
	gantry_crane.Command := IDLE;
	CraneIsReady := FALSE;
END_PROGRAM

PROGRAM _CYCLIC
	(* Insert code here *)
	CASE EmergencyStopMachine OF
		0: IF EmergencyStop AND State <> EmergencyState THEN
				State := EmergencyState;
				gantry_crane.Command := EMERGENCY_STOP_REQUEST;
				box_crane.Command := EMERGENCY_STOP_REQUEST;
				EmergencyStopMachine := 1;
			END_IF
		1: IF NOT EmergencyStop THEN
				EmergencyStopMachine := 0;
			END_IF
	END_CASE

	CASE ImmediateStopMachine OF
		0: IF ImmediateStop AND State <> ImmediateStopState THEN
				OldState := State;
				OldBoxCraneCommand := box_crane.Command;
				OldGantryCraneCommand := gantry_crane.Command;
				OldPositionBoxCraneGoal := box_crane_goal;
				OldPositionGantryCraneGoal := gantry_crane_goal;
				box_crane.Command := IMMEDIATE_STOP_REQUEST;
				gantry_crane.Command := IMMEDIATE_STOP_REQUEST;
				State := ImmediateStopState;
				ImmediateStopMachine := 1;
			END_IF
		1: IF NOT ImmediateStop THEN
				ImmediateStopMachine := 0;
			END_IF
	END_CASE

	CASE State OF

		EmergencyState:
			IF NOT EmergencyStop THEN
				gantry_crane.Command := IDLE;
				box_crane.Command := IDLE;
				CraneIsReady := FALSE;
				CraneEnable := FALSE;
				State := Idle;
			END_IF

		ImmediateStopState:
			IF NOT ImmediateStop AND CraneStart THEN
				CraneStart := FALSE;
				State := OldState;
				box_crane.Command := OldBoxCraneCommand;
				box_crane_goal := OldPositionBoxCraneGoal;

				gantry_crane.Command := OldGantryCraneCommand;
				gantry_crane_goal := OldPositionGantryCraneGoal;
			END_IF

		Idle:
			IF CraneEnable THEN
				// Abbassare il Box_Crane
				slide_rail_right_disable_request := TRUE;
				pusher_x_disable_request := TRUE;
				pusher_z_disable_request := TRUE;
				vacuum_box_crane_disable_request := TRUE;
				cardboard_disable_request := TRUE;
				CounterFloor := 0;

				IF box_crane_AXIS <> BOX_CRANE_HOMING_POSITION THEN
					box_crane_goal := BOX_CRANE_HOMING_POSITION;
					box_crane.Command := CHANGE_POSITION;
				END_IF
				IF gantry_crane_AXIS <> GANTRY_CRANE_HOMING_POSITION THEN
					gantry_crane_goal := GANTRY_CRANE_HOMING_POSITION;
					gantry_crane.Command := CHANGE_POSITION;
				END_IF
				State := CardBoardPickHoming;
			END_IF

		CardBoardPickHoming:
			IF 	(slide_rail_right_disable_request = FALSE AND pusher_x_disable_request = FALSE AND pusher_z_disable_request = FALSE
				AND BoxCranePositionReached AND GantryCranePositionReached) THEN
				IF box_crane_AXIS <> CARDBOARD_PICK_POSITION THEN
					box_crane_goal := CARDBOARD_PICK_POSITION;
					box_crane.Command := CHANGE_POSITION;
				END_IF
				State := CardBoardVacuum;
			END_IF

		CardBoardVacuum:
			IF BoxCranePositionReached  THEN
				cardboard_enable_request := TRUE;
				vacuum_box_crane_enable_request := TRUE;
				State := CardBoardVacuumHoming;
			END_IF

		CardBoardVacuumHoming:
			IF (vacuum_box_crane_enable_request = FALSE  AND cardboard_enable_request = FALSE) THEN
				cardboard_disable_request := TRUE;
				IF box_crane_AXIS <> BOX_CRANE_HOMING_POSITION THEN
					box_crane_goal := BOX_CRANE_HOMING_POSITION;
					box_crane.Command := CHANGE_POSITION;
					State := Homing;
				END_IF
			END_IF

		Homing:
			IF  BoxCranePositionReached AND cardboard_disable_request = FALSE THEN
				CraneIsReady := TRUE;
				CraneEnable := FALSE;
				State := HomingDone;
			END_IF

		HomingDone:
			// crane ready, wait for start
			IF CraneStart THEN
				CraneStart := FALSE;
				CraneIsReady := FALSE;
				CounterFloor := CounterFloor + 1;
				slide_rail_right_enable_request := TRUE;
				pusher_z_enable_request := TRUE;
				State := MoveToCardBoardPositioning;
			END_IF

		MoveToCardBoardPositioning:
			IF slide_rail_right_enable_request = FALSE  AND pusher_z_enable_request = FALSE THEN // the closure of the slide_rail_right should be defined in correspondance of the MAIN-FEEDER-CRANE interface
				IF (CounterFloor MOD 2 = 1) = TRUE THEN
					IF box_crane_AXIS <> BOX_CRANE_FLOOR1_POSITION THEN
						box_crane_goal := BOX_CRANE_FLOOR1_POSITION;
						box_crane.Command := CHANGE_POSITION;
					END_IF
				ELSE
					IF box_crane_AXIS <> BOX_CRANE_FLOOR2_POSITION THEN
						box_crane_goal := BOX_CRANE_FLOOR2_POSITION;
						box_crane.Command := CHANGE_POSITION;
					END_IF
				END_IF
				IF gantry_crane_AXIS <> GANTRY_CRANE_CARDBOARD_POSITION THEN
					gantry_crane_goal := GANTRY_CRANE_CARDBOARD_POSITION;
					gantry_crane.Command := CHANGE_POSITION;
				END_IF

				IF NOT (BoxCranePositionReached AND GantryCranePositionReached) THEN
					State := CardBoardPositioning;
				END_IF
			END_IF

		CardBoardPositioning:
			IF  (BoxCranePositionReached AND GantryCranePositionReached) THEN
				vacuum_box_crane_disable_request := TRUE;
				State := MoveToPallet;
			END_IF

		MoveToPallet:
			IF (vacuum_box_crane_disable_request = FALSE) THEN
				IF gantry_crane_AXIS <> GANTRY_CRANE_PALLET_POSITION THEN
					gantry_crane_goal := GANTRY_CRANE_PALLET_POSITION;
					gantry_crane.Command := CHANGE_POSITION;
				END_IF
				State := FreeBoxes;
			END_IF

		FreeBoxes:
			IF GantryCranePositionReached THEN
				slide_rail_right_disable_request := TRUE;
				IF (CounterFloor MOD 2 = 1) = TRUE THEN
					State := MoveToCardBoardBuffer1;
				ELSE
					State := MoveToCardBoardBuffer2_1;
				END_IF
			END_IF

		MoveToCardBoardBuffer1:
			IF slide_rail_right_disable_request = FALSE THEN
				pusher_x_enable_request := TRUE; // POTREBBE ESSERE NECESSARIO FARE PRIMA LA RICHIESTA E POI MUOVERE IL CRANE
				IF box_crane_AXIS <> CARDBOARD_PICK_POSITION THEN
					box_crane_goal := CARDBOARD_PICK_POSITION;
					box_crane.Command := CHANGE_POSITION;
				END_IF
				IF gantry_crane_AXIS <> GANTRY_CRANE_HOMING_POSITION THEN
					gantry_crane_goal := GANTRY_CRANE_HOMING_POSITION;
					gantry_crane.Command := CHANGE_POSITION;
				END_IF
				State := CardBoardPick;
			END_IF

		MoveToCardBoardBuffer2_1:
			IF slide_rail_right_disable_request = FALSE THEN
				pusher_x_enable_request := TRUE; // POTREBBE ESSERE NECESSARIO FARE PRIMA LA RICHIESTA E POI MUOVERE IL CRANE
				IF gantry_crane_AXIS <> GANTRY_CRANE_HOMING_POSITION THEN
					gantry_crane_goal := GANTRY_CRANE_HOMING_POSITION;
					gantry_crane.Command := CHANGE_POSITION;
				END_IF
				State := MoveToCardBoardBuffer2_2;
			END_IF
		MoveToCardBoardBuffer2_2:
			IF pusher_x_enable_request = FALSE AND GantryCranePositionReached THEN
				IF box_crane_AXIS <> CARDBOARD_PICK_POSITION THEN
					box_crane_goal := CARDBOARD_PICK_POSITION;
					box_crane.Command := CHANGE_POSITION;
				END_IF
				State := CardBoardPick;
			END_IF

		CardBoardPick:
			IF pusher_x_enable_request = FALSE AND BoxCranePositionReached AND GantryCranePositionReached THEN
				cardboard_enable_request := TRUE;
				vacuum_box_crane_enable_request := TRUE;
				State := MoveToHomingPosition;
			END_IF

		MoveToHomingPosition:
			IF vacuum_box_crane_enable_request = FALSE AND cardboard_enable_request = FALSE THEN
				IF box_crane_AXIS <> BOX_CRANE_HOMING_POSITION THEN
					box_crane_goal := BOX_CRANE_HOMING_POSITION;
					box_crane.Command := CHANGE_POSITION;
				END_IF
				cardboard_disable_request := TRUE;
				pusher_x_disable_request := TRUE;
				pusher_z_disable_request := TRUE;
				State := CheckForHomingDone;
			END_IF

		CheckForHomingDone:
			IF pusher_x_disable_request = FALSE AND pusher_z_disable_request = FALSE AND cardboard_disable_request = FALSE AND BoxCranePositionReached AND GantryCranePositionReached THEN
				State := HomingDone;
				CraneIsReady := TRUE;
			END_IF

	END_CASE

	// Device Calls
	// Generic Axis
	box_crane.NewSetPoint := box_crane_goal;
	box_crane.DeviceTimer := box_crane_timer; // if elapsed gives fault (See GenericAxis library)
	box_crane.ActualPosition := box_crane_AXIS;
	box_crane.TGT_SENSOR := TRUE;
	box_crane();
	box_crane_TGT_POS := box_crane.TargetPosition;
	BoxCranePositionReached := box_crane.InPosition;

	gantry_crane.NewSetPoint := gantry_crane_goal;
	gantry_crane.DeviceTimer := gantry_crane_timer; // if elapsed gives fault (See GenericAxis library)
	gantry_crane.ActualPosition := gantry_crane_AXIS;
	gantry_crane.TGT_SENSOR := TRUE;
	gantry_crane();
	gantry_crane_TGT_POS := gantry_crane.TargetPosition;
	GantryCranePositionReached := gantry_crane.InPosition;

	// Generic Device
	pusher_x.DeviceOperation := OperationType;
	pusher_x.DeviceClock := TRUE;
	pusher_x.DeviceDiagnosticsEnabled := TRUE;
	pusher_x.DeviceEnablePreset := FALSE;
	pusher_x.DeviceEnableTime := pusher_x_enable_time;
	pusher_x.DeviceDisableTime := pusher_x_disable_time;
	pusher_x.DeviceType := DEVICE_WITHOUT_FEEDBACK OR DEVICE_WITH_SINGLE_ACTUATION;
	pusher_x(DeviceEnableRequest := pusher_x_enable_request, DeviceDisableRequest := pusher_x_disable_request);
	pusher_x_EN := pusher_x.EnableDevice;

	pusher_z.DeviceOperation := OperationType;
	pusher_z.DeviceClock := TRUE;
	pusher_z.DeviceDiagnosticsEnabled := TRUE;
	pusher_z.DeviceEnablePreset := FALSE;
	pusher_z.DeviceEnableTime := pusher_z_enable_time;
	pusher_z.DeviceDisableTime := pusher_z_disable_time;
	pusher_z.DeviceType := DEVICE_WITHOUT_FEEDBACK OR DEVICE_WITH_SINGLE_ACTUATION;
	pusher_z(DeviceEnableRequest := pusher_z_enable_request, DeviceDisableRequest := pusher_z_disable_request);
	pusher_z_EN := pusher_z.EnableDevice;

	slide_rail_right.DeviceOperation := OperationType;
	slide_rail_right.DeviceClock := TRUE;
	slide_rail_right.DeviceDiagnosticsEnabled := TRUE;
	slide_rail_right.DeviceEnablePreset := FALSE;
	slide_rail_right.DeviceEnableTime := slide_rail_right_enable_time;
	slide_rail_right.DeviceDisableTime := slide_rail_right_disable_time;
	slide_rail_right.DeviceType := DEVICE_WITHOUT_FEEDBACK OR DEVICE_WITH_SINGLE_ACTUATION;
	slide_rail_right(DeviceEnableRequest := slide_rail_right_enable_request, DeviceDisableRequest := slide_rail_right_disable_request);
	slide_rail_right_EN := slide_rail_right.EnableDevice;

	vacuum_box_crane.DeviceOperation := OperationType;
	vacuum_box_crane.DeviceClock := TRUE;
	vacuum_box_crane.DeviceDiagnosticsEnabled := TRUE;
	vacuum_box_crane.DeviceEnablePreset := FALSE;
	vacuum_box_crane.DeviceEnableTime := vacuum_box_crane_enable_time;
	vacuum_box_crane.DeviceDisableTime := vacuum_box_crane_disable_time;
	vacuum_box_crane.DeviceEnabledSensor := vacuum_box_crane_VACUUM;
	vacuum_box_crane.DeviceType := DEVICE_WITH_ENABLE_FEEDBACK OR DEVICE_WITH_SINGLE_ACTUATION;
	vacuum_box_crane(DeviceEnableRequest := vacuum_box_crane_enable_request, DeviceDisableRequest := vacuum_box_crane_disable_request);
	vacuum_box_crane_GRIP := vacuum_box_crane.EnableDevice;

	cardboard.DeviceOperation := OperationType;
	cardboard.DeviceClock := TRUE;
	cardboard.DeviceDiagnosticsEnabled := TRUE;
	cardboard.DeviceEnablePreset := FALSE;
	cardboard.DeviceEnableTime := cardboard_enable_time;
	cardboard.DeviceDisableTime := cardboard_disable_time;
	cardboard.DeviceType := DEVICE_WITHOUT_FEEDBACK OR DEVICE_WITH_SINGLE_ACTUATION;
	cardboard(DeviceEnableRequest := cardboard_enable_request, DeviceDisableRequest := cardboard_disable_request);
	cardboard_TRIG := cardboard.EnableDevice;

	// Signals

	(* Pusher X *)
	PusherXActuatorFaultE := pusher_x.DeviceActuatorFault;
	PusherXDisableSensorFaultE := pusher_x.DeviceDisabledSensorFault;
	PusherXEnableSensorFaultE := pusher_x.DeviceEnabledSensorFault;

	(* Pusher Z *)
	PusherZActuatorFaultE := pusher_z.DeviceActuatorFault;
	PusherZDisableSensorFaultE := pusher_z.DeviceDisabledSensorFault;
	PusherZEnableSensorFaultE := pusher_z.DeviceEnabledSensorFault;

	(* Slide Rail Right *)
	SlideRailRightActuatorFaultE := slide_rail_right.DeviceActuatorFault;
	SlideRailRightDisableFaultE := slide_rail_right.DeviceDisabledSensorFault;
	SlideRailRightEnableFaultE := slide_rail_right.DeviceEnabledSensorFault;

	(* Vacuum Box Crane *)
	VacuumBoxCraneActuatorFaultE := vacuum_box_crane.DeviceActuatorFault;
	VacuumBoxCraneDisableFaultE := vacuum_box_crane.DeviceDisabledSensorFault;
	VacuumBoxCraneEnableFaultE := vacuum_box_crane.DeviceEnabledSensorFault;

	(* Cardboard *)
	CardboardActuatorFaultE := cardboard.DeviceActuatorFault;
	CardboardDisableFaultE := cardboard.DeviceDisabledSensorFault;
	CardboardEnableFaultE := cardboard.DeviceEnabledSensorFault;

	(* Box Crane *)
	BoxCraneFaultSignalE :=  box_crane.DeviceFault;

	(* Gantry Crane *)
	GantryCraneFaultSignalE := gantry_crane.DeviceFault;

END_PROGRAM

PROGRAM _EXIT
	(* Insert code here *)

END_PROGRAM
```

### Program Logical/PalletHandlerMachine (IEC)

#### Types.typ
```iecst
TYPE
	StateType :
		(
		Idle,
		Homing,
		HomingDone,
		MoveToPalletPositioning,
		ReleasePallet,
		MoveToNewPallet,
		GraspPallet,
		RaisePalletStack,
		MoveConveyor,
		PalletApproach,
		PalletSlowdown,
		PalletArrived,
		PalletStop,
		EmergencyState,
		StopState,
		ImmediateStopState
		);
END_TYPE
```

#### Variables.var
```iecst
(*pallet_lifter*)
VAR
	pallet_lifter : GenericAxis;
END_VAR
VAR CONSTANT
	PALLET_LIFTER_IDLE : REAL := 0.0;
	PALLET_LIFTER_RELEASE : REAL := -0.258;
	PALLET_LIFTER_GRASP : REAL := -0.12;
END_VAR
VAR
	PalletLifterPositionReached : BOOL;
	pallet_lifter_goal : REAL;
END_VAR
VAR CONSTANT
	pallet_lifter_timer : INT := 200;
END_VAR
(*pallet_fork*)
VAR
	pallet_fork : GenericDevice_FB;
END_VAR
VAR CONSTANT
	pallet_fork_enable_time : INT := 200;
	pallet_fork_disable_time : INT := 20;
END_VAR
VAR
	pallet_fork_enable_request : BOOL;
	pallet_fork_disable_request : BOOL;
END_VAR
(*pallet_conveyor_1*)
VAR
	pallet_conveyor_1 : GenericDevice_FB;
END_VAR
VAR CONSTANT
	pallet_conveyor_1_enable_time : INT := 5;
	pallet_conveyor_1_disable_time : INT := 5;
END_VAR
VAR
	pallet_conveyor_1_enable_request : BOOL;
	pallet_conveyor_1_disable_reques : BOOL;
END_VAR
(*pallet_conveyor_2*)
VAR
	pallet_conveyor_2 : GenericAxis;
	pallet_conveyor_2_velocity : REAL;
END_VAR
VAR CONSTANT
	LOW_VELOCITY : REAL := 0.1;
	FAST_VELOCITY : REAL := 0.5;
	STANDSTILL : REAL := 0.0;
END_VAR
VAR
	PalletConveyor2VelReached : BOOL;
	pallet_conveyor_2_timer : INT;
	State : StateType;
	EmergencyStopMachine : INT;
	OldState : StateType;
	ImmediateStopMachine : INT;
	SuspendDevices : BOOL;
	OldPalletConveyor2Command : WORD;
	OldPalletLifterCommand : WORD;
	OldPositionPalletLifterGoal : REAL;
	OldPositionPalletConv2Vel : REAL;
END_VAR
```

#### Main.st
```iecst
// PALLET HANDLER MACHINE
// INTERFACE
// 	INPUT:
// 		PalletHandlerEnable : BOOL : It enables the machine and executes the Homing if it is not already done.
//		PalletHandlerStart : BOOL : It starts a machine cycle if The machine is Ready
//		PalletHandlerStop : BOOL
//		PalletHandlerEmergencyStop : BOOL
//
//	OUTPUT:
//		PalletHandlerIsEnable : BOOL : True if the machine is ready to start a new cycle.
//		PalletHandlerIsReady : BOOL : True if the machine is ready to start a new cycle.
//		PalletHandlerIsStop : BOOL
//		PalletHandlerIsStopEmergency : BOOL

PROGRAM _INIT
	(* Insert code here *)
	State := Idle;
	pallet_conveyor_2.Command := IDLE;
	pallet_lifter.Command := IDLE;

END_PROGRAM

PROGRAM _CYCLIC
	(* Insert code here *)
	CASE EmergencyStopMachine OF
		0: IF EmergencyStop AND State <> EmergencyState THEN
				State := EmergencyState;
				pallet_lifter.Command := EMERGENCY_STOP_REQUEST;
				pallet_conveyor_2.Command := EMERGENCY_STOP_REQUEST;
				EmergencyStopMachine := 1;
			END_IF
		1: IF NOT EmergencyStop THEN
				EmergencyStopMachine := 0;
			END_IF
	END_CASE

	CASE ImmediateStopMachine OF
		0: IF ImmediateStop AND State <> ImmediateStopState THEN
				OldState := State;
				SuspendDevices := TRUE;
				OldPalletLifterCommand := pallet_lifter.Command;
				OldPalletConveyor2Command := pallet_conveyor_2.Command;
				OldPositionPalletLifterGoal := pallet_lifter_goal;
				OldPositionPalletConv2Vel := pallet_conveyor_2_velocity;
				pallet_lifter.Command := IMMEDIATE_STOP_REQUEST;
				pallet_conveyor_2.Command := IMMEDIATE_STOP_REQUEST;
				State := ImmediateStopState;
				ImmediateStopMachine := 1;
			END_IF
		1: IF NOT ImmediateStop THEN
				ImmediateStopMachine := 0;
			END_IF
	END_CASE

	CASE State OF
		EmergencyState:
			IF NOT EmergencyStop THEN
				State := Idle;
				PalletHandlerIsReady := FALSE;
				PalletHandlerEnable := FALSE;
				pallet_lifter.Command := IDLE;
				pallet_conveyor_2.Command := IDLE;
			END_IF

		ImmediateStopState:
			IF NOT ImmediateStop AND PalletHandlerStart THEN
				PalletHandlerStart := FALSE;
				SuspendDevices := FALSE;
				State := OldState;
				pallet_lifter.Command := OldPalletLifterCommand;
				pallet_lifter_goal := OldPositionPalletLifterGoal;

				pallet_conveyor_2.Command := OldPalletConveyor2Command;
				pallet_conveyor_2_velocity := OldPositionPalletConv2Vel;
			END_IF

		Idle:
			IF PalletHandlerEnable THEN				// da impostare la variabile
				pallet_fork_disable_request := TRUE;
				pallet_conveyor_1_disable_reques := TRUE;
				IF pallet_lifter_TGT_POS <> PALLET_LIFTER_IDLE THEN
					pallet_lifter_goal := PALLET_LIFTER_IDLE;
					pallet_lifter.Command := CHANGE_POSITION;
				END_IF
				IF pallet_conveyor_2_ACT_VEL <> STANDSTILL THEN
					pallet_conveyor_2.Command := CHANGE_VELOCITY;
					pallet_conveyor_2_velocity := STANDSTILL;
				END_IF
				State := Homing;
			END_IF

		Homing:
			IF pallet_fork_disable_request = FALSE AND pallet_conveyor_1_disable_reques = FALSE AND PalletLifterPositionReached AND PalletConveyor2VelReached THEN
				State := HomingDone;
				PalletHandlerIsReady := TRUE;
				PalletHandlerEnable := FALSE;
			END_IF

		HomingDone:
			IF PalletHandlerStart THEN
				PalletHandlerStart := FALSE;
				PalletHandlerIsReady := FALSE;
				IF pallet_lifter_TGT_POS <> PALLET_LIFTER_RELEASE THEN
					pallet_lifter_goal := PALLET_LIFTER_RELEASE;
					pallet_lifter.Command := CHANGE_POSITION;
				END_IF
				IF pallet_conveyor_2_ACT_VEL <> FAST_VELOCITY THEN
					pallet_conveyor_2.Command := CHANGE_VELOCITY;
					pallet_conveyor_2_velocity := FAST_VELOCITY;
				END_IF
				State := MoveToPalletPositioning;
			END_IF

		MoveToPalletPositioning:
			IF PalletLifterPositionReached AND 	PalletConveyor2VelReached THEN
				pallet_fork_enable_request := TRUE;
				State := ReleasePallet;
			END_IF

		ReleasePallet:
			IF pallet_fork_enable_request = FALSE THEN
				IF pallet_lifter_TGT_POS <> PALLET_LIFTER_GRASP THEN
					pallet_lifter_goal := PALLET_LIFTER_GRASP;
					pallet_lifter.Command := CHANGE_POSITION;
				END_IF
				State := MoveToNewPallet;
			END_IF

		MoveToNewPallet:
			IF PalletLifterPositionReached THEN
				pallet_fork_disable_request := TRUE;
				State := GraspPallet;
			END_IF

		GraspPallet:
			IF pallet_fork_disable_request = FALSE THEN
				IF pallet_lifter_TGT_POS <> PALLET_LIFTER_IDLE THEN
					pallet_lifter_goal := PALLET_LIFTER_IDLE;
					pallet_lifter.Command := CHANGE_POSITION;
				END_IF
				State := RaisePalletStack;
			END_IF

		RaisePalletStack:
			IF PalletLifterPositionReached THEN
				pallet_conveyor_1_enable_request := TRUE;
				State := MoveConveyor;
			END_IF

		MoveConveyor:
			IF pallet_conveyor_1_enable_request = FALSE THEN
				State := PalletApproach;
			END_IF

		PalletApproach:
			IF pallet_light_barrier2_enabled THEN
				pallet_conveyor_1_disable_reques := TRUE;
				IF pallet_conveyor_2_ACT_VEL <> LOW_VELOCITY THEN
					pallet_conveyor_2.Command := CHANGE_VELOCITY;
					pallet_conveyor_2_velocity := LOW_VELOCITY;
				END_IF
				State := PalletSlowdown;
			END_IF

		PalletSlowdown:
			IF pallet_conveyor_1_disable_reques = FALSE AND	PalletConveyor2VelReached THEN
				State := PalletArrived;
			END_IF

		PalletArrived:
			IF pallet_light_barrier_enabled THEN
				IF pallet_conveyor_2_ACT_VEL <> STANDSTILL THEN
					pallet_conveyor_2.Command := CHANGE_VELOCITY;
					pallet_conveyor_2_velocity := STANDSTILL;
				END_IF
				State := PalletStop;
			END_IF

		PalletStop:
			IF PalletConveyor2VelReached THEN
				PalletHandlerIsReady := TRUE;
				State := HomingDone;
			END_IF

	END_CASE

	// pallet_fork
	pallet_fork.DeviceOperation := OperationType;
	pallet_fork.DeviceClock := TRUE;
	pallet_fork.DeviceDiagnosticsEnabled := TRUE;
	pallet_fork.DeviceEnablePreset := FALSE;
	pallet_fork.DeviceEnableTime := pallet_fork_enable_time;
	pallet_fork.DeviceDisableTime := pallet_fork_disable_time;
	pallet_fork.DeviceEnabledSensor := pallet_fork_left_FB;
	pallet_fork.DeviceType := DEVICE_WITH_ENABLE_FEEDBACK OR DEVICE_WITH_SINGLE_ACTUATION;
	pallet_fork(DeviceEnableRequest := pallet_fork_enable_request, DeviceDisableRequest := pallet_fork_disable_request);
	pallet_fork_left_EN := pallet_fork.EnableDevice;

	// pallet_conveyor_1
	pallet_conveyor_1.DeviceOperation := OperationType;
	pallet_conveyor_1.DeviceClock := TRUE;
	pallet_conveyor_1.DeviceDiagnosticsEnabled := TRUE;
	pallet_conveyor_1.ImmediateStop := SuspendDevices OR EmergencyStop;
	pallet_conveyor_1.DeviceEnablePreset := FALSE;
	pallet_conveyor_1.DeviceEnableTime := pallet_conveyor_1_enable_time;
	pallet_conveyor_1.DeviceDisableTime := pallet_conveyor_1_disable_time;
	pallet_conveyor_1.DeviceType := DEVICE_WITHOUT_FEEDBACK OR DEVICE_WITH_SINGLE_ACTUATION OR DEVICE_IMMEDIATE_STOP_AUTOMATIC;
	pallet_conveyor_1(DeviceEnableRequest := pallet_conveyor_1_enable_request, DeviceDisableRequest := pallet_conveyor_1_disable_reques);
	pallet_conveyor_1_FWD := pallet_conveyor_1.EnableDevice;

	// pallet_lifter
	pallet_lifter.NewSetPoint := pallet_lifter_goal;
	pallet_lifter.DeviceTimer := pallet_lifter_timer; // if elapsed gives fault (See GenericAxis library)
	pallet_lifter.ActualPosition := pallet_lifter_AXIS;
	pallet_lifter.TGT_SENSOR := TRUE;
	pallet_lifter();
	pallet_lifter_TGT_POS := pallet_lifter.TargetPosition;
	PalletLifterPositionReached := pallet_lifter.InPosition;

	// pallet_conveyor_2
	pallet_conveyor_2.NewSetPoint := pallet_conveyor_2_velocity;
	pallet_conveyor_2.DeviceTimer := pallet_conveyor_2_timer; // if elapsed gives fault (See GenericAxis library)
	pallet_conveyor_2.ActualVelocity := pallet_conveyor_2_ACT_VEL;
	pallet_conveyor_2.TGT_SENSOR := TRUE;
	pallet_conveyor_2();
	pallet_conveyor_2_ACT_VEL := pallet_conveyor_2.TargetVelocity;
	PalletConveyor2VelReached := pallet_conveyor_2.InVelocity;

	// Signals

	(* Pallet Fork *)
	PalletForkActuatorFaultE := pallet_fork.DeviceActuatorFault;
	PalletForkDisableSensorFaultE := pallet_fork.DeviceDisabledSensorFault;
	PalletForkEnableSensorFaultE := pallet_fork.DeviceEnabledSensorFault;

	(* Pallet Lifter *)
	PalletLifterFaultSignalE := pallet_lifter.DeviceFault;

	(* Pallet Conveyor 1 *)
	PalletConv1ActuatorFaultE := pallet_conveyor_1.DeviceActuatorFault;
	PalletConv1DisableSensorFaultE := pallet_conveyor_1.DeviceDisabledSensorFault;
	PalletConv1SensorFaultE := pallet_conveyor_1.DeviceEnabledSensorFault;

	(* Pallet Conveyor 2 *)
	PalletConv2FaultSignalE := pallet_conveyor_2.DeviceFault;

END_PROGRAM

PROGRAM _EXIT
	(* Insert code here *)

END_PROGRAM
```

### Program Logical/InputBridge (IEC)

#### Main.st
```iecst
PROGRAM _INIT
	(* Insert code here *)

END_PROGRAM

PROGRAM _CYCLIC
	// Feeder input variable simulation establishment
	laser_sensor_IR := ComTCP_SimInputs.laser_sensor_IR;
	laser_sensor_2_IR := ComTCP_SimInputs.laser_sensor2_IR;
	carriage_2_AXIS := ComTCP_SimInputs.carriage_2_AXIS;
	carriage_2_RCHD := ComTCP_SimInputs.carriage_2_RCHD;
	pusher_LBK := ComTCP_SimInputs.pusher_LBK;
	pusher_LFR := ComTCP_SimInputs.pusher_LFR;
	turnpusher_LBK := NOT(ComTCP_SimInputs.turnpusher_LBK);
	turnpusher_LFR := NOT(ComTCP_SimInputs.turnpusher_LFR);

	// Crane input variable simulation establishment
	vacuum_box_crane_VACUUM := ComTCP_SimInputs.vaccum_box_crane_VACUUM;
	box_crane_AXIS := ComTCP_SimInputs.box_crane_AXIS;
	gantry_crane_AXIS := ComTCP_SimInputs.gantry_crane_AXIS;

	// Pallet Handler input variable simulation establishment
	pallet_lifter_AXIS := ComTCP_SimInputs.pallet_lifter_AXIS;
	pallet_fork_left_FB := ComTCP_SimInputs.pallet_fork_left_FB;
	pallet_light_barrier_1_IR := ComTCP_SimInputs.pallet_light_barrier_1_IR;
	pallet_light_barrier_2_IR := ComTCP_SimInputs.pallet_light_barrier_2_IR;

END_PROGRAM

PROGRAM _EXIT
	(* Insert code here *)

END_PROGRAM
```

### Program Logical/OutputBridge (IEC)

#### Main.st
```iecst
PROGRAM _INIT
	(* Insert code here *)

END_PROGRAM

PROGRAM _CYCLIC
	// Feeder output variable simulation establishment
	ComTCP_SimOutputs.conveyor_if_FWD := conveyor_if_FWD;
	ComTCP_SimOutputs.conveyer_turn1_FWD :=  conveyor_turn1_FWD;
	ComTCP_SimOutputs.conveyer_end_FWD := conveyor_end_FWD;
	ComTCP_SimOutputs.pusher_FW := pusher_FW;
	ComTCP_SimOutputs.turnpusher_BWD := NOT(turnpusher_BWD);
	ComTCP_SimOutputs.turnpusher_FWD := NOT(turnpusher_FWD);
	ComTCP_SimOutputs.carriage_2_TGT_POS := carrige_2_TGT_POS;

	// Crane output variable simulation establishment
	ComTCP_SimOutputs.vaccum_box_crane_GRIP := vacuum_box_crane_GRIP;
	ComTCP_SimOutputs.gantry_crane_TGT_POS := gantry_crane_TGT_POS;
	ComTCP_SimOutputs.box_crane_TGT_POS := box_crane_TGT_POS;
	ComTCP_SimOutputs.cartboard_TRIG := cardboard_TRIG;
	ComTCP_SimOutputs.slide_rail_right_EN := slide_rail_right_EN;
	ComTCP_SimOutputs.pusher_z_EN := pusher_z_EN;
	ComTCP_SimOutputs.pusher_x_EN := pusher_x_EN;

	// Pallet Handler output variable simulation establishment
	ComTCP_SimOutputs.pallet_lifter_TGT_POS := pallet_lifter_TGT_POS;
	ComTCP_SimOutputs.pallet_fork_left_EN := pallet_fork_left_EN;
	ComTCP_SimOutputs.pallet_conveyor_1_FWD := pallet_conveyor_1_FWD;
	ComTCP_SimOutputs.pallet_conveyor_2_ACT_VEL := pallet_conveyor_2_ACT_VEL;

END_PROGRAM

PROGRAM _EXIT
	(* Insert code here *)

END_PROGRAM
```

- Visualisation Logical/mappView (not shown)

### Program Logical/MainControl (IEC)

#### Types.typ
```iecst
TYPE
	StateType :
		(
		FeedBoxes,
		HomingDone,
		Homing,
		Idle,
		WaitForBoxes,
		WaitForPush,
		FeederPush,
		BoxOnPalletPositioning,
		WaitBoxesOnPallet,
		ChangePallet,
		WaitForNewPallet,
		EmergencyState,
		CheckActivationsFromStop,
		ImmediateStopState,
		StopState
		);
END_TYPE
```

#### Variables.var
```iecst
VAR
	State : StateType;
	CounterFloor : INT;
	OldState : StateType;
	ImmediateStopMachine : INT;
	EmergencyStopMachine : INT;
	OnPhaseStopMachine : INT;
END_VAR
```

#### Main.st
```iecst
// MAIN CONTROL MACHINE
// http://localhost:81/index.html?visuId=vis_0
// INTERFACE
// 	INPUT:
// 		MainEnable : BOOL : It enables the machine and executes the Homing if it is not already done.
//		MainStart : BOOL : It starts a machine cycle if The machine is Ready
//		MainStop : BOOL
//		MainEmergencyStop : BOOL
//
//	OUTPUT:
//		MainIsEnable : BOOL : True if the machine is ready to start a new cycle.
//		MainIsReady : BOOL : True if the machine is ready to start a new cycle.
//		MainIsStop : BOOL
//		MainIsStopEmergency : BOOL

PROGRAM _INIT
	(* Insert code here *)
	State := Idle;
	MainEnable := FALSE;
	MainStart := FALSE;
	CounterFloor := 0;
	CounterPallet := 0;
END_PROGRAM

PROGRAM _CYCLIC
	(* Insert code here *)
	CASE EmergencyStopMachine OF
		0: IF EmergencyStop AND State <> EmergencyState THEN
				State := EmergencyState;
				MainEnable := FALSE;
				MainStart := FALSE;
				EmergencyStopMachine := 1;
			END_IF
		1: IF NOT EmergencyStop THEN
				EmergencyStopMachine := 0;
				MainEnable := FALSE;
				MainStart := FALSE;
			END_IF
	END_CASE

	CASE ImmediateStopMachine OF
		0: IF ImmediateStop AND State <> ImmediateStopState THEN
				OldState := State;
				State := ImmediateStopState;
				MainEnable := FALSE;
				MainStart := FALSE;
				ImmediateStopMachine := 1;
			END_IF
		1: IF NOT ImmediateStop THEN
				ImmediateStopMachine := 0;
				MainEnable := FALSE;
				MainStart := FALSE;
				OperationType := ENABLED;
			END_IF
	END_CASE

	CASE OnPhaseStopMachine OF
		0: IF OnPhaseStop THEN
				OnPhaseStopPerforming := TRUE;
				OnPhaseStopMachine := 1;
			END_IF
		1: IF NOT OnPhaseStop THEN
				OnPhaseStopMachine := 0;
			END_IF
	END_CASE

	CASE State OF
		EmergencyState:
			IF NOT EmergencyStop THEN
				State := Idle;
				MainEnable := FALSE;
				MainStart := FALSE;
				OperationType := INIT;
			END_IF

		ImmediateStopState:
			IF MainStart AND NOT ImmediateStop THEN
				MainStart := FALSE;
				FeederStart := TRUE;
				CraneStart := TRUE;
				PalletHandlerStart := TRUE;
				State := CheckActivationsFromStop;
			END_IF

		CheckActivationsFromStop:
			IF FeederStart = FALSE AND CraneStart = FALSE AND PalletHandlerStart = FALSE THEN
				State := OldState;
				OperationType := RUN;
			END_IF

		Idle:
			CounterPallet := 0;
			OnPhaseStopPerforming := FALSE;
			IF MainEnable THEN
				CounterFloor := 0;
				OperationType := ENABLED;
				FeederEnable := TRUE;
				CraneEnable := TRUE;
				PalletHandlerEnable := TRUE;
				State := Homing;
			END_IF

		Homing:
			IF FeederEnable = FALSE AND CraneEnable = FALSE AND PalletHandlerEnable = FALSE THEN // AND PalletEnable ...
				MainEnable := FALSE;
				MainStart := FALSE;
				State := HomingDone;
			END_IF

		HomingDone:
			IF OnPhaseStopPerforming THEN
				OnPhaseStopPerforming := FALSE;
			END_IF

			IF MainStart THEN
				OperationType := RUN;
				MainStart := FALSE;
				FeederStart := TRUE;
				PalletHandlerStart := TRUE;
				State := FeedBoxes;
			END_IF

		FeedBoxes:
			IF FeederStart = FALSE THEN
				State := WaitForBoxes; // Push of the Boxes
			END_IF

		WaitForBoxes:
			IF FeederIsReady = TRUE AND CraneIsReady = TRUE THEN
				FeederStart := TRUE;
				State := FeederPush;
				CounterFloor := CounterFloor + 1;
			END_IF

		FeederPush:
			IF FeederStart = FALSE THEN
				State := WaitForPush;
			END_IF

		WaitForPush:
			IF FeederIsReady = TRUE AND CraneIsReady = TRUE THEN // AND PalletHandler
				IF NOT (OnPhaseStop AND (CounterFloor MOD 2 <> 1) = TRUE) THEN
					FeederStart := TRUE; // Boxes accumulation
				END_IF

				CraneStart := TRUE;
				State := BoxOnPalletPositioning;
			END_IF

		BoxOnPalletPositioning:
			IF FeederStart = FALSE AND CraneStart = FALSE THEN
				State := WaitBoxesOnPallet;
			END_IF

		WaitBoxesOnPallet:
			IF CraneIsReady = TRUE AND PalletHandlerIsReady = TRUE THEN
				IF (CounterFloor MOD 2 <> 1) = TRUE AND NOT OnPhaseStop THEN
					PalletHandlerStart := TRUE;
					CounterPallet := CounterPallet +1;
					State := ChangePallet;
				ELSIF (CounterFloor MOD 2 <> 1) = TRUE AND OnPhaseStop THEN
					State := HomingDone;
					OnPhaseStopPerforming := FALSE;
					MainStart := FALSE;
					CounterPallet := CounterPallet +1;
					OperationType := ENABLED;
				ELSE
					State := WaitForBoxes;
				END_IF

			END_IF

		ChangePallet:
			IF PalletHandlerStart = FALSE AND CraneStart = FALSE  THEN
				State := WaitForNewPallet;
			END_IF

		WaitForNewPallet:
			IF PalletHandlerIsReady = TRUE THEN
				State := WaitForBoxes;
			END_IF
	END_CASE;

END_PROGRAM

PROGRAM _EXIT
	(* Insert code here *)

END_PROGRAM
```

### Program Logical/SignalManager (IEC)

#### Variables.var
```iecst
VAR
	SignalManagement : SignalManagement_FB;
	SignalOutputs : DWORD;
END_VAR
VAR CONSTANT
	mPusherXActuatorFault : INT := 1;
	mPusherXDisableSensorFault : INT := 2;
	mPusherXEnableSensorFault : INT := 3;
	mPusherZActuatorFault : INT := 4;
	mPusherZDisableSensorFault : INT := 5;
	mPusherZEnableSensorFault : INT := 6;
	mSlideRailRightActuatorFault : INT := 7;
	mSlideRailRightDisableFault : INT := 8;
	mSlideRailRightEnableFault : INT := 9;
	mVacuumBoxCraneActuatorFault : INT := 10;
	mVacuumBoxCraneDisableFault : INT := 11;
	mVacuumBoxCraneEnableFault : INT := 12;
	mCardboardActuatorFault : INT := 13;
	mCardboardDisableFault : INT := 14;
	mCardboardEnableFault : INT := 15;
	mBoxCraneFaultSignal : INT := 16;
	mGantryCraneFaultSignal : INT := 17;
	mPusherActuatorFault : INT := 18;
	mPusherDisableSensorFault : INT := 19;
	mPusherEnableSensorFault : INT := 20;
	mConveyorIfActuatorFault : INT := 21;
	mConveyorIfDisableSensorFault : INT := 22;
	mConveyorIfEnableSensorFault : INT := 23;
	mConveyorTurn1ActuatorFault : INT := 24;
	mConveyorTurn1DisableSensorFault : INT := 25;
	mConveyorTurn1EnableSensorFault : INT := 26;
	mConveyorEndActuatorFault : INT := 27;
	mConveyorEndDisableSensorFault : INT := 28;
	mConveyorEndEnableSensorFault : INT := 29;
	mCarriagePositionFaultSignal : INT := 30;
	mPalletForkActuatorFault : INT := 31;
	mPalletForkDisableSensorFault : INT := 32;
	mPalletForkEnableSensorFault : INT := 33;
	mPalletLifterFaultSignal : INT := 34;
	mPalletConv1ActuatorFault : INT := 35;
	mPalletConv1DisableSensorFault : INT := 36;
	mPalletConv1SensorFault : INT := 37;
	mPalletConv2FaultSignal : INT := 38;
	mTurnpusherActuatorFault : INT := 39;
	mTurnpusherDisableSensorFault : INT := 40;
	mTurnpusherEnableSensorFault : INT := 41;
	mImmediateStopButton : INT := 42;
	mEmergencyStopButton : INT := 43;
	mOnPhaseStopButton : INT := 44;
END_VAR
```

#### Main.st
```iecst
PROGRAM _INIT
	(* Insert code here *)
END_PROGRAM

PROGRAM _CYCLIC
	(* Insert code here *)

	IF OperationType = INIT THEN
		SignalManagement(OperationType := START_CONFIGURATION);
		SignalManagement.OperationType := CONFIGURATION;
	ELSE
		SignalManagement(OperationType := START_GENERATION);
		SignalManagement.OperationType := GENERATION;
		SignalManagement.Reset := ResetButton;
	END_IF

	(* IMMEDIATE STOP *)

	(* IMMEDIATE STOP *)
	SignalManagement(SignalType := ALARM OR DISPLAY_LOG,
	SignalCode := mImmediateStopButton,
	SignalOutput := IMMEDIATE_STOP,
	InputString := 'IMMEDIATE STOP ACTIVATED',
	ActivationSignal := ImmediateStopButton);

	(* EMERGENCY STOP *)
	SignalManagement(SignalType := ALARM OR DISPLAY_LOG,
	SignalCode := mEmergencyStopButton,
	SignalOutput := EMERGENCY_STOP,
	InputString := 'EMERGENCY STOP ACTIVATED',
	ActivationSignal := EmergencyStopButton);

	(* ON PHASE STOP *)
	SignalManagement(SignalType := INFORMATION OR DISPLAY_LOG,
	SignalCode := mOnPhaseStopButton,
	SignalOutput := ON_PHASE_STOP,
	InputString := 'ON PHASE STOP PERFORMING ...',
	ActivationSignal := OnPhaseStopPerforming OR OnPhaseStopButton);

	(* CRANE MACHINE *)

	(* Pusher X *)
	SignalManagement(SignalType := ALARM OR DISPLAY_LOG,
	SignalCode := mPusherXActuatorFault,
	SignalOutput := EMERGENCY_STOP,
	InputString := 'Pusher_X Actuator Fault',
	ActivationSignal := PusherXActuatorFaultE);

	SignalManagement(SignalType := ALARM OR DISPLAY_LOG,
	SignalCode := mPusherXDisableSensorFault,
	SignalOutput := EMERGENCY_STOP,
	InputString := 'Pusher_X Disable Sensor Fault',
	ActivationSignal := PusherXDisableSensorFaultE);

	SignalManagement(SignalType := ALARM OR DISPLAY_LOG,
	SignalCode := mPusherXEnableSensorFault,
	SignalOutput := EMERGENCY_STOP,
	InputString := 'Pusher_X Enable Sensor Fault',
	ActivationSignal := PusherXEnableSensorFaultE);

	(* Pusher Z *)
	SignalManagement(SignalType := ALARM OR DISPLAY_LOG,
	SignalCode := mPusherZActuatorFault,
	SignalOutput := EMERGENCY_STOP,
	InputString := 'Pusher_Z Actuator Fault',
	ActivationSignal := PusherZActuatorFaultE);

	SignalManagement(SignalType := ALARM OR DISPLAY_LOG,
	SignalCode := mPusherZDisableSensorFault,
	SignalOutput := EMERGENCY_STOP,
	InputString := 'Pusher_Z Disable Sensor Fault',
	ActivationSignal := PusherZDisableSensorFaultE);

	SignalManagement(SignalType := ALARM OR DISPLAY_LOG,
	SignalCode := mPusherZEnableSensorFault,
	SignalOutput := EMERGENCY_STOP,
	InputString := 'Pusher_Z Enable Sensor Fault',
	ActivationSignal := PusherZEnableSensorFaultE);

	(* Slide Rail Right *)
	SignalManagement(SignalType := ALARM OR DISPLAY_LOG,
	SignalCode := mSlideRailRightActuatorFault,
	SignalOutput := EMERGENCY_STOP,
	InputString := 'Slide Rail Right Actuator Fault',
	ActivationSignal := SlideRailRightActuatorFaultE);

	SignalManagement(SignalType := ALARM OR DISPLAY_LOG,
	SignalCode := mSlideRailRightDisableFault,
	SignalOutput := EMERGENCY_STOP,
	InputString := 'Slide Rail Right Disable Sensor Fault',
	ActivationSignal := SlideRailRightDisableFaultE);

	SignalManagement(SignalType := ALARM OR DISPLAY_LOG,
	SignalCode := mSlideRailRightEnableFault,
	SignalOutput := EMERGENCY_STOP,
	InputString := 'Slide Rail Right Enable Sensor Fault',
	ActivationSignal := SlideRailRightEnableFaultE);

	(* Vacuum Box Crane *)
	SignalManagement(SignalType := ALARM OR DISPLAY_LOG,
	SignalCode := mVacuumBoxCraneActuatorFault,
	SignalOutput := EMERGENCY_STOP,
	InputString := 'Vacuum Box Crane Actuator Fault',
	ActivationSignal := VacuumBoxCraneActuatorFaultE OR SimVacuumBoxCraneActuatorFaultE);

	SignalManagement(SignalType := ALARM OR DISPLAY_LOG,
	SignalCode := mVacuumBoxCraneDisableFault,
	SignalOutput := EMERGENCY_STOP,
	InputString := 'Vacuum Box Crane Disable Sensor Fault',
	ActivationSignal := VacuumBoxCraneDisableFaultE);

	SignalManagement(SignalType := ALARM OR DISPLAY_LOG,
	SignalCode := mVacuumBoxCraneEnableFault,
	SignalOutput := EMERGENCY_STOP,
	InputString := 'Vacuum Box Crane Enable Sensor Fault',
	ActivationSignal := VacuumBoxCraneEnableFaultE);

	(* Cardboard *)
	SignalManagement(SignalType := ALARM OR DISPLAY_LOG,
	SignalCode := mCardboardActuatorFault,
	SignalOutput := EMERGENCY_STOP,
	InputString := 'Cardboard Actuator Fault',
	ActivationSignal := CardboardActuatorFaultE);

	SignalManagement(SignalType := ALARM OR DISPLAY_LOG,
	SignalCode := mCardboardDisableFault,
	SignalOutput := EMERGENCY_STOP,
	InputString := 'Cardboard Disable Sensor Fault',
	ActivationSignal := CardboardDisableFaultE);

	SignalManagement(SignalType := ALARM OR DISPLAY_LOG,
	SignalCode := mCardboardEnableFault,
	SignalOutput := EMERGENCY_STOP,
	InputString := 'Cardboard Enable Sensor Fault',
	ActivationSignal := CardboardEnableFaultE);

	(* Box Crane *)
	SignalManagement(SignalType := ALARM OR DISPLAY_LOG,
	SignalCode := mBoxCraneFaultSignal,
	SignalOutput := EMERGENCY_STOP,
	InputString := 'Box Crane Fault',
	ActivationSignal := BoxCraneFaultSignalE OR SimBoxCraneFaultSignalE);

	(* Gantry Crane *)
	SignalManagement(SignalType := ALARM OR DISPLAY_LOG,
	SignalCode := mGantryCraneFaultSignal,
	SignalOutput := EMERGENCY_STOP,
	InputString := 'Gantry Crane Fault',
	ActivationSignal := GantryCraneFaultSignalE);

	(* FEEDER *)

	(* Turnpusher *)
	SignalManagement(SignalType := ALARM OR DISPLAY_LOG,
	SignalCode := mTurnpusherActuatorFault,
	SignalOutput := EMERGENCY_STOP,
	InputString := 'Turnpusher Actuator Fault',
	ActivationSignal := TurnpusherActuatorFaultE);

	SignalManagement(SignalType := ALARM OR DISPLAY_LOG,
	SignalCode := mTurnpusherDisableSensorFault,
	SignalOutput := EMERGENCY_STOP,
	InputString := 'Turnpusher Disable Sensor Fault',
	ActivationSignal := TurnpusherDisableSensorFaultE);

	SignalManagement(SignalType := ALARM OR DISPLAY_LOG,
	SignalCode := mTurnpusherEnableSensorFault,
	SignalOutput := EMERGENCY_STOP,
	InputString := 'Turnpusher Enable Sensor Fault',
	ActivationSignal := TurnpusherEnableSensorFaultE);

	(* Pusher *)
	SignalManagement(SignalType := ALARM OR DISPLAY_LOG,
	SignalCode := mPusherActuatorFault,
	SignalOutput := EMERGENCY_STOP,
	InputString := 'Pusher Actuator Fault',
	ActivationSignal := PusherActuatorFaultE OR SimPusherActuatorFaultE);

	SignalManagement(SignalType := ALARM OR DISPLAY_LOG,
	SignalCode := mPusherDisableSensorFault,
	SignalOutput := EMERGENCY_STOP,
	InputString := 'Pusher Disable Sensor Fault',
	ActivationSignal := PusherDisableSensorFaultE OR SimPusherDisableSensorFaultE);

	SignalManagement(SignalType := ALARM OR DISPLAY_LOG,
	SignalCode := mPusherEnableSensorFault,
	SignalOutput := EMERGENCY_STOP,
	InputString := 'Pusher Enable Sensor Fault',
	ActivationSignal := PusherEnableSensorFaultE);

	(* Conveyor If *)
	SignalManagement(SignalType := ALARM OR DISPLAY_LOG,
	SignalCode := mConveyorIfActuatorFault,
	SignalOutput := EMERGENCY_STOP,
	InputString := 'Conveyor If Actuator Fault',
	ActivationSignal := ConveyorIfActuatorFaultE);

	SignalManagement(SignalType := ALARM OR DISPLAY_LOG,
	SignalCode := mConveyorIfDisableSensorFault,
	SignalOutput := EMERGENCY_STOP,
	InputString := 'Conveyor If Disable Sensor Fault',
	ActivationSignal := ConveyorIfDisableSensorFaultE);

	SignalManagement(SignalType := ALARM OR DISPLAY_LOG,
	SignalCode := mConveyorIfEnableSensorFault,
	SignalOutput := EMERGENCY_STOP,
	InputString := 'Conveyor If Enable Sensor Fault',
	ActivationSignal := ConveyorIfEnableSensorFaultE);

	(* Conveyor Turn1 *)
	SignalManagement(SignalType := ALARM OR DISPLAY_LOG,
	SignalCode := mConveyorTurn1ActuatorFault,
	SignalOutput := EMERGENCY_STOP,
	InputString := 'Conveyor Turn1 Actuator Fault',
	ActivationSignal := ConveyorTurn1ActuatorFaultE);

	SignalManagement(SignalType := ALARM OR DISPLAY_LOG,
	SignalCode := mConveyorTurn1DisableSensorFault,
	SignalOutput := EMERGENCY_STOP,
	InputString := 'Conveyor Turn1 Disable Sensor Fault',
	ActivationSignal := ConveyorTurn1DisableSensorFaultE);

	SignalManagement(SignalType := ALARM OR DISPLAY_LOG,
	SignalCode := mConveyorTurn1EnableSensorFault,
	SignalOutput := EMERGENCY_STOP,
	InputString := 'Conveyor Turn1 Enable Sensor Fault',
	ActivationSignal := ConveyorTurn1EnableSensorFaultE);

	(* Conveyor End *)
	SignalManagement(SignalType := ALARM OR DISPLAY_LOG,
	SignalCode := mConveyorEndActuatorFault,
	SignalOutput := EMERGENCY_STOP,
	InputString := 'Conveyor End Actuator Fault',
	ActivationSignal := ConveyorEndActuatorFaultE);

	SignalManagement(SignalType := ALARM OR DISPLAY_LOG,
	SignalCode := mConveyorEndDisableSensorFault,
	SignalOutput := EMERGENCY_STOP,
	InputString := 'Conveyor End Disable Sensor Fault',
	ActivationSignal := ConveyorEndDisableSensorFaultE);

	SignalManagement(SignalType := ALARM OR DISPLAY_LOG,
	SignalCode := mConveyorEndEnableSensorFault,
	SignalOutput := EMERGENCY_STOP,
	InputString := 'Conveyor End Enable Sensor Fault',
	ActivationSignal := ConveyorEndEnableSensorFaultE);

	(* Carriage *)
	SignalManagement(SignalType := ALARM OR DISPLAY_LOG,
	SignalCode := mCarriagePositionFaultSignal,
	SignalOutput := EMERGENCY_STOP,
	InputString := 'Carriage Position Fault',
	ActivationSignal := CarriagePositionFaultSignalE);

	(* PALLET HANDLER *)

	(* Pallet Fork *)
	SignalManagement(SignalType := ALARM OR DISPLAY_LOG,
	SignalCode := mPalletForkActuatorFault,
	SignalOutput := EMERGENCY_STOP,
	InputString := 'Pallet Fork Actuator Fault',
	ActivationSignal := PalletForkActuatorFaultE OR SimPalletForkActuatorFaultE);

	SignalManagement(SignalType := ALARM OR DISPLAY_LOG,
	SignalCode := mPalletForkDisableSensorFault,
	SignalOutput := EMERGENCY_STOP,
	InputString := 'Pallet Fork Disable Sensor Fault',
	ActivationSignal := PalletForkDisableSensorFaultE);

	SignalManagement(SignalType := ALARM OR DISPLAY_LOG,
	SignalCode := mPalletForkEnableSensorFault,
	SignalOutput := EMERGENCY_STOP,
	InputString := 'Pallet Fork Enable Sensor Fault',
	ActivationSignal := PalletForkEnableSensorFaultE OR SimPalletForkEnableSensorFaultE);

	(* Pallet Lifter *)
	SignalManagement(SignalType := ALARM OR DISPLAY_LOG,
	SignalCode := mPalletLifterFaultSignal,
	SignalOutput := EMERGENCY_STOP,
	InputString := 'Pallet Lifter Fault',
	ActivationSignal := PalletLifterFaultSignalE);

	(* Pallet Conveyor 1 *)
	SignalManagement(SignalType := ALARM OR DISPLAY_LOG,
	SignalCode := mPalletConv1ActuatorFault,
	SignalOutput := EMERGENCY_STOP,
	InputString := 'Pallet Conveyor 1 Actuator Fault',
	ActivationSignal := PalletConv1ActuatorFaultE);

	SignalManagement(SignalType := ALARM OR DISPLAY_LOG,
	SignalCode := mPalletConv1DisableSensorFault,
	SignalOutput := EMERGENCY_STOP,
	InputString := 'Pallet Conveyor 1 Disable Sensor Fault',
	ActivationSignal := PalletConv1DisableSensorFaultE);

	SignalManagement(SignalType := ALARM OR DISPLAY_LOG,
	SignalCode := mPalletConv1SensorFault,
	SignalOutput := EMERGENCY_STOP,
	InputString := 'Pallet Conveyor 1 Sensor Fault',
	ActivationSignal := PalletConv1SensorFaultE);

	(* Pallet Conveyor 2 *)
	SignalManagement(SignalType := ALARM OR DISPLAY_LOG,
	SignalCode := mPalletConv2FaultSignal,
	SignalOutput := EMERGENCY_STOP,
	InputString := 'Pallet Conveyor 2 Fault',
	ActivationSignal := PalletConv2FaultSignalE);

	IF OperationType <> INIT THEN
		SignalManagement(OperationType := MESSAGES_GENERATION);
		LogFile := SignalManagement.LogFile;
		MainMessage := SignalManagement.MainMessage;
		SignalOutputs := SignalManagement.SignalOutputs;
		EmergencyStop := (SignalOutputs AND EMERGENCY_STOP) = EMERGENCY_STOP;
		ImmediateStop := (SignalOutputs AND IMMEDIATE_STOP) = IMMEDIATE_STOP;
		OnPhaseStop := (SignalOutputs AND ON_PHASE_STOP) = ON_PHASE_STOP;
	END_IF

	ResetEnable := SignalManagement.ResetEnable;
	ResetButton := FALSE;
	ImmediateStopButton := FALSE;
	EmergencyStopButton := FALSE;
	OnPhaseStopButton := FALSE;

END_PROGRAM

PROGRAM _EXIT
	(* Insert code here *)

END_PROGRAM
```

### Program Logical/InputFilter (IEC)

#### Variables.var
```iecst
VAR
	Laser1Filter : filter_FB;
	Laser2Filter : filter_FB;
	palletLightBarrier1Filter : filter_FB;
	palletLightBarrier2Filter : filter_FB;
END_VAR
```

#### Main.st
```iecst
PROGRAM _INIT
	(* Insert code here *)

END_PROGRAM

PROGRAM _CYCLIC
	(* Insert code here *)

	Laser1Filter.Clock := TRUE;
	Laser1Filter.ActivationDelay := 0;
	Laser1Filter.DeactivationDelay := 10;
	Laser1Filter.Signal := laser_sensor_IR;
	Laser1Filter(OperationType := OperationType);
	laser_sensor_IR_enabled := Laser1Filter.DelayedSignal;

	Laser2Filter.Clock := TRUE;
	Laser2Filter.ActivationDelay := 0;
	Laser2Filter.DeactivationDelay := 3;
	Laser2Filter.Signal := laser_sensor_2_IR;
	Laser2Filter(OperationType := OperationType);
	laser_sensor_2_IR_enabled := Laser2Filter.DelayedSignal;

	palletLightBarrier1Filter.Clock := TRUE;
	palletLightBarrier1Filter.ActivationDelay := 0;
	palletLightBarrier1Filter.DeactivationDelay := 10;
	palletLightBarrier1Filter.Signal := pallet_light_barrier_1_IR;
	palletLightBarrier1Filter(OperationType := OperationType);
	pallet_light_barrier_enabled := palletLightBarrier1Filter.DelayedSignal;

	palletLightBarrier2Filter.Clock := TRUE;
	palletLightBarrier2Filter.ActivationDelay := 0;
	palletLightBarrier2Filter.DeactivationDelay := 5;
	palletLightBarrier2Filter.Signal := pallet_light_barrier_2_IR;
	palletLightBarrier2Filter(OperationType := OperationType);
	pallet_light_barrier2_enabled := palletLightBarrier2Filter.DelayedSignal;

END_PROGRAM

PROGRAM _EXIT
	(* Insert code here *)

END_PROGRAM
```

### Program Logical/InterfaceHandler (IEC)

#### Variables.var
```iecst
VAR
	Counter : INT;
END_VAR
```

#### Main.st
```iecst
PROGRAM _INIT
	(* Insert code here *)
	Counter := 10;
END_PROGRAM

PROGRAM _CYCLIC
	(* Insert code here *)

	IF Counter = 0 THEN
		Counter := 10;
	ELSE
		Counter := Counter -1;
	END_IF

	CASE OperationType OF
		INIT:
			OperationTypeString := 'INIT';
			IF Counter = 0 THEN
				BlueLight := NOT BlueLight;
			END_IF
			GreenLight := FALSE;

		ENABLED:
			OperationTypeString := 'ENABLED';
			BlueLight := TRUE;
			IF Counter = 0 THEN
				GreenLight := NOT GreenLight;
			END_IF

		RUN:
			OperationTypeString := 'RUN';
			GreenLight := TRUE;
			BlueLight := FALSE;

		STOP:
			OperationTypeString := 'STOP';
			GreenLight := FALSE;
			BlueLight := FALSE;

	END_CASE

	IF OnPhaseStop THEN
		OrangeLight := TRUE;
	ELSE
		OrangeLight := FALSE;
	END_IF

	IF ImmediateStop THEN
		YellowLight := TRUE;
	ELSE
		YellowLight := FALSE;
	END_IF

	IF EmergencyStop THEN
		RedLight := TRUE;
	ELSE
		RedLight := FALSE;
	END_IF

	IF ResetEnable AND Counter = 0 THEN
		WhiteLight := NOT WhiteLight;
	ELSIF NOT ResetEnable THEN
		WhiteLight := FALSE;
	END_IF

	IF HomeButton THEN
		InfoCarousel := 'content_0';
	END_IF

	IF ErrorButton THEN
		InfoCarousel := 'content_1';
	END_IF

END_PROGRAM

PROGRAM _EXIT
	(* Insert code here *)

END_PROGRAM
```

Listed in the project but not available here: Logical/Global.typ, Logical/Libraries/ComTCP, Logical/Libraries/Signal_lib/Types.typ, Logical/Libraries/Filter/Types.typ, Logical/Libraries/Filter/Constants.var, Logical/MNG_Package.typ, Logical/MNG_Package.var
